// TwinCAT 3 PLC project PML_Base_Library
// Title: PML_Base_Library
// Company: SPT
// ProjectVersion: 0.1
// ProgramVersion: 3.1.4023.0
// libraries:
//   Tc2_Standard, * (Beckhoff Automation GmbH)
//   Tc2_System, * (Beckhoff Automation GmbH)
//   Tc3_EventLogger, * (Beckhoff Automation GmbH)
//   Tc3_PackML_V2, * (Beckhoff Automation GmbH)
// project tree:
//   Base/01_PML/01_Module/01_Base/01_GVL/ GVL_PML_Base.TcGVL
//   Base/01_PML/01_Module/01_Base/02_DUT/01_ENUM/ E_AlarmResponse.TcDUT, E_PMLUnitMode.TcDUT
//   Base/01_PML/01_Module/01_Base/02_DUT/02_STRUCT/ ST_PMLModuleBase_HMI.TcDUT, ST_PMLModuleBase_VISU.TcDUT, ST_PMLSubUnitInfoExt.TcDUT
//   Base/01_PML/01_Module/01_Base/03_ITFs/ ITF_PMLControl.TcIO, ITF_PMLModuleBase.TcIO
//   Base/01_PML/01_Module/01_Base/ FB_PMLModuleBase.TcPOU
//   Base/01_PML/01_Module/02_Events/ FB_PMLModeLogger.TcPOU, FB_PMLStateLogger.TcPOU
//   Base/01_PML/01_Module/03_PMLControl/03_ITFs/ ITF_PackML_ExternalControl.TcIO, ITF_PackML_ExternalControl_Simplified.TcIO
//   Base/01_PML/01_Module/03_PMLControl/ FB_ModuleExternalCommandControl.TcPOU, FB_PackML_ExternalControl.TcPOU, FB_PackML_PushButtonControl.TcPOU
//   Base/01_PML/01_Module/05_Visualizations/ V_MachineModule.TcVIS, V_Module.TcVIS
//   Base/01_PML/99_Templates/ FB_Module_TEMPLATE.TcPOU
//   Base/02_Component/ FB_ComponentBase.TcPOU, ITF_ComponentBase.TcIO, ST_ComponentBase_HMI.TcDUT
//   Base/03_Utilities/01_Events/ F_CreateAllEventsInClass.TcPOU, F_GetMaxSeverityRaised.TcPOU, F_RaiseAlarmAndSetFlags.TcPOU, F_RaiseAlarmWithStringParameters.TcPOU, F_RaiseAlarmWithStringsAndFlags.TcPOU
//   Base/03_Utilities/02_DataStructures/01_Tree/01_Tree_IndexBased/ FB_Tree_IndexBased.TcPOU, ITF_Tree_IndexBased.TcIO, ST_Tree_IndexBased_Node.TcDUT
//   Base/03_Utilities/02_DataStructures/02_FIFO/ FB_FIFO_ULINT_Array.TcPOU
//   Base/03_Utilities/03_Math/01_LREAL/ F_LREAL_RoundToPlace.TcPOU
//   / GlobalTextList.TcGTLO, Visualization Manager.TcVMO (not stored)

// ---- Base/01_PML/01_Module/01_Base/02_DUT/01_ENUM/E_AlarmResponse.TcDUT
{attribute 'qualified_only'}
{attribute 'strict'}
TYPE E_AlarmResponse :
(
	Abort_ImmediateError,
	Abort_Immediate,
	Stop_Immediate,
	Stop_Controlled,
	Hold_Immediate,
	Hold_Controlled,	
	Suspend_Immediate,
	Suspend_Controlled,
	NoResponse	
);
END_TYPE

// ---- Base/01_PML/01_Module/01_Base/02_DUT/01_ENUM/E_PMLUnitMode.TcDUT
{attribute 'qualified_only'}		//Note that this is not "Strict" since it needs to interact with the mode manager, which uses DINTs for mode
TYPE E_PMLUnitMode:
(
	ePMLUnitMode_Invalid 		:= 0,
	ePMLUnitMode_Production		:= 1,
	ePMLUnitMode_Maintenance	:= 2,
	ePMLUnitMode_Manual			:= 3
	// User defined modes
    (*ePMLUnitMode_SemiAutomatic  :=  4,
    ePMLUnitMode_DryRun         :=  5,
	ePMLUnitMode_Standalone		:=  6,
	ePMLUnitMode_Usermode4		:=  7,
	ePMLUnitMode_Usermode5 		:=  8,
	ePMLUnitMode_Usermode6 		:=  9,
	ePMLUnitMode_Usermode7 		:=  10 *)	
) DINT;
END_TYPE

// ---- Base/01_PML/01_Module/01_Base/02_DUT/02_STRUCT/ST_PMLModuleBase_HMI.TcDUT
TYPE ST_PMLModuleBase_HMI :
STRUCT
	bEnabled							: BOOL;					//Enables or disables the packml Machine of the module (prevents the module from going past idle)
	eMode								: E_PMLUnitMode;		//Current UnitMode of the module
	nModuleID							: UDINT;				//Unique identifying number for the module
	sModuleName							: STRING;				//Human-readable module name for user-side messaging
	eState								: Tc3_PackML_V2.E_PMLState;
	bLogStateChanges 					: BOOL := TRUE; 		//Toggle to permit or suppress state change logging (Should be tied to HMI setting to optionally reduce event logger clutter)
	bLogModeChanges 					: BOOL := TRUE; 		//Toggle to permit or suppress state change logging (Should be tied to HMI setting to optionally reduce event logger clutter)
	
	//Control information
	bHMIControlAvailable				: BOOL;		//Set TRUE *FROM PLC* when HMI requests can be processed
	bIncomingHMIRequest 				: BOOL;		//Pulses TRUE when an HMI request is issued
	bHMICommandConfirmation				: BOOL;		//Confirms receipt and subsequent processing of the command sent by the HMI
	
	bModeCommandHMIRequest				: BOOL;		//Pulses TRUE when an HMI mode change request is issued
	bStateCommandHMIRequest				: BOOL;		//Pulses TRUE when an HMI state change request is issued
	bEnableHMIRequest					: BOOL;		//HMI requests to enable the module
	bDisableHMIRequest 					: BOOL;		//HMI requests to disable the module
	bActivateStateLogHMIRequest			: BOOL;		//HMI requests to enable the module
	bDeactivateStateLogHMIRequest 		: BOOL;		//HMI requests to disable the module
	bActivateModeLogHMIRequest			: BOOL;		//HMI requests to enable the module
	bDeactivateModeLogHMIRequest 		: BOOL;		//HMI requests to disable the module
	eModeCommandHMIValue				: E_PMLUnitMode;
	eStateCommandHMIValue				: Tc3_PackML_V2.E_PMLCommand;
	a_sModeNames						: ARRAY[0..31] OF STRING;
	
END_STRUCT
END_TYPE

// ---- Base/01_PML/01_Module/01_Base/02_DUT/02_STRUCT/ST_PMLModuleBase_VISU.TcDUT
TYPE ST_PMLModuleBase_VISU :
STRUCT
	bEnabled			: BOOL;					//Enables or disables the packml Machine of the module (prevents the module from going past idle)
	eMode				: E_PMLUnitMode;		//Current UnitMode of the module
	nModuleID			: UDINT;					//Unique identifying number for the module
	sModuleName			: STRING;				//Human-readable module name for user-side messaging
	eState				: Tc3_PackML_V2.E_PMLState;
	
	//eModeCommandValue	: E_PMLUnitMode;
	///eStateCommandValue	: Tc3_PackML_V2.E_PMLCommand;
	bStartPressed		: BOOL;
	///bStartEnabled		: BOOL;
	bStopPressed		: BOOL;
	///bStopEnabled		: BOOL;
	bResetPressed		: BOOL;
	///bResetEnabled		: BOOL;
	bClearPressed		: BOOL;
	///bClearEnabled		: BOOL;	
	
	bAbortPressed		: BOOL;
	bHoldPressed		: BOOL;
	bUnholdPressed		: BOOL;
	bSuspendPressed		: BOOL;
	bUnsuspendPressed	: BOOL;
	
	// Mode things
	bProductionPressed	: BOOL;
	bMaintenancePressed	: BOOL;
	bManualPressed		: BOOL;
	
END_STRUCT
END_TYPE

// ---- Base/01_PML/01_Module/01_Base/02_DUT/02_STRUCT/ST_PMLSubUnitInfoExt.TcDUT
TYPE ST_PMLSubUnitInfoExt EXTENDS ST_PMLSubUnitInfo :	//Extended Struct of ST_PMLSubUnitInfo
STRUCT
	nModuleID 						: DINT; 				//Machine ID for messaging and Identification
	sModuleName						: STRING;				//Human readable machine name for messaging
	UnitModeCurrent					: E_PMLProtectedUnitMode;
	ActiveAlarm						: BOOL;
END_STRUCT
END_TYPE

// ---- Base/02_Component/ST_ComponentBase_HMI.TcDUT
TYPE ST_ComponentBase_HMI :
STRUCT
	//Status information
	bEnabled	: BOOL;
	bSimulate 	: BOOL;
	sName		: STRING;
	bActive		: BOOL;
	bError		: BOOL;
	nErrorID	: UDINT;
	
	//Control information
	bHMIControlAvailable	: BOOL;		//Set TRUE *FROM PLC* when HMI requests can be processed
	bIncomingHMIRequest 	: BOOL;		//Pulses TRUE when an HMI request is issued
	bHMICommandConfirmation	: BOOL;		//Confirms receipt and subsequent processing of the command sent by the HMI
	
	bEnableHMIRequest				: BOOL;		//HMI requests to enable the component
	bDisableHMIRequest 				: BOOL;		//HMI requests to disable the component
	bSimulateOperationHMIRequest 	: BOOL;		//HMI requests to change the component to simulation mode
	bStandardOperationHMIRequest	: BOOL;		//HMI requests to change the component to standard mode
	bResetHMIRequest				: BOOL;		//HMI requests to reset the component
	
END_STRUCT
END_TYPE

// ---- Base/03_Utilities/02_DataStructures/01_Tree/01_Tree_IndexBased/ST_Tree_IndexBased_Node.TcDUT
TYPE ST_Tree_IndexBased_Node :
STRUCT
	sName 		: STRING;
	nChildCount	: DINT;
	nParent		: DINT;
	a_nChildren	: ARRAY[0..15] OF DINT;
	nDepth		: DINT;
END_STRUCT
END_TYPE

// ---- Base/01_PML/01_Module/01_Base/01_GVL/GVL_PML_Base.TcGVL
///{attribute 'qualified_only'}
VAR_GLOBAL CONSTANT
	MAX_NO_OF_SUBMODULES			: UDINT := 20;
	MAX_NO_OF_COMPONENTS			: UDINT := 32;

	ePMLUNITMODEDEFAULT			: E_PMLUnitMode := E_PMLUnitMode.ePMLUnitMode_Production;
	ePMLSTATEDEFAULT			: E_PMLCommand := E_PMLCommand.ePMLCommand_Abort;

END_VAR

// ---- Base/01_PML/01_Module/01_Base/03_ITFs/ITF_PMLControl.TcIO
INTERFACE ITF_PMLControl

PROPERTY Mode : E_PMLUnitMode
GET
END_GET
END_PROPERTY

PROPERTY ModeCommand : DINT
SET
END_SET
END_PROPERTY

PROPERTY State : E_PMLState
GET
END_GET
END_PROPERTY

PROPERTY StateCommand : E_PMLCommand
SET
END_SET
END_PROPERTY

END_INTERFACE

// ---- Base/01_PML/01_Module/01_Base/03_ITFs/ITF_PMLModuleBase.TcIO
INTERFACE ITF_PMLModuleBase EXTENDS ITF_PMLControl

PROPERTY AncestorIDs : STRING
GET
END_GET
SET
END_SET
END_PROPERTY

PROPERTY CurrentAlarmSeverity :  TcEventSeverity
GET
END_GET
END_PROPERTY

METHOD CyclicLogic
END_METHOD

PROPERTY Enabled : BOOL
GET
END_GET
SET
END_SET
END_PROPERTY

PROPERTY LogModeChanges : BOOL
GET
END_GET
SET
END_SET
END_PROPERTY

PROPERTY LogStateChanges : BOOL
GET
END_GET
SET
END_SET
END_PROPERTY

PROPERTY MasterDataStructure_Adder :  ITF_Tree_IndexBased
GET
END_GET
SET
END_SET
END_PROPERTY

PROPERTY ModuleID : UDINT
GET
END_GET
SET
END_SET
END_PROPERTY

PROPERTY ModuleName : STRING
GET
END_GET
SET
END_SET
END_PROPERTY

PROPERTY ParentResponse_Critical : E_AlarmResponse
GET
END_GET
SET
END_SET
END_PROPERTY

PROPERTY ParentResponse_Error : E_AlarmResponse
GET
END_GET
SET
END_SET
END_PROPERTY

PROPERTY ParentResponse_Warning : E_AlarmResponse
GET
END_GET
SET
END_SET
END_PROPERTY

PROPERTY ParentResponseDef : ARRAY[0..4] OF E_AlarmResponse
GET
END_GET
SET
END_SET
END_PROPERTY

PROPERTY SimulateAllChildren : BOOL
GET
END_GET
SET
END_SET
END_PROPERTY

END_INTERFACE

// ---- Base/01_PML/01_Module/03_PMLControl/03_ITFs/ITF_PackML_ExternalControl.TcIO
INTERFACE ITF_PackML_ExternalControl EXTENDS ITF_PackML_ExternalControl_Simplified

PROPERTY Mode : DINT
GET
END_GET
SET
END_SET
END_PROPERTY

PROPERTY ModeCommand : DINT
GET
END_GET
SET
END_SET
END_PROPERTY

PROPERTY ModeCommandPulse : BOOL
GET
END_GET
SET
END_SET
END_PROPERTY

PROPERTY State : E_PMLState
GET
END_GET
SET
END_SET
END_PROPERTY

PROPERTY StateCommand : E_PMLCommand
GET
END_GET
SET
END_SET
END_PROPERTY

PROPERTY StateCommandPulse : BOOL
GET
END_GET
SET
END_SET
END_PROPERTY

END_INTERFACE

// ---- Base/01_PML/01_Module/03_PMLControl/03_ITFs/ITF_PackML_ExternalControl_Simplified.TcIO
INTERFACE ITF_PackML_ExternalControl_Simplified


PROPERTY ClearEnabled : BOOL
GET
END_GET
SET
END_SET
END_PROPERTY


PROPERTY ClearPressed : BOOL
GET
END_GET
SET
END_SET
END_PROPERTY

PROPERTY ResetEnabled : BOOL
GET
END_GET
SET
END_SET
END_PROPERTY

PROPERTY ResetPressed : BOOL
GET
END_GET
SET
END_SET
END_PROPERTY

PROPERTY StartEnabled : BOOL
GET
END_GET
SET
END_SET
END_PROPERTY

PROPERTY StartPressed : BOOL
GET
END_GET
SET
END_SET
END_PROPERTY

PROPERTY StopEnabled : BOOL
GET
END_GET
SET
END_SET
END_PROPERTY

PROPERTY StopPressed : BOOL
GET
END_GET
SET
END_SET
END_PROPERTY

END_INTERFACE

// ---- Base/02_Component/ITF_ComponentBase.TcIO
INTERFACE ITF_ComponentBase

PROPERTY Active : BOOL	//TRUE when the component is in motion or otherwise completing a commanded task
GET
END_GET
END_PROPERTY

METHOD AllowHMIControl : BOOL
VAR_INPUT
END_VAR
END_METHOD

METHOD BlockHMIControl : BOOL
VAR_INPUT
END_VAR
END_METHOD

PROPERTY CurrentAlarmSeverity : TcEventSeverity
GET
END_GET
END_PROPERTY

METHOD CyclicLogic : BOOL		//Should be called Externally akin to the PML Modules
END_METHOD

PROPERTY Enabled : BOOL	//Enables or disables the component
GET
END_GET
SET
END_SET
END_PROPERTY

PROPERTY Error : BOOL	//Boolean to signal that an error has ocurred
GET
END_GET
END_PROPERTY

PROPERTY ErrorID : UDINT	//Integer ID to identify the proper alarm to be posted from the parent module
GET
END_GET
SET
END_SET
END_PROPERTY

PROPERTY Name : STRING
GET
END_GET
SET
END_SET
END_PROPERTY

PROPERTY ParentResponseDefinitions : ARRAY[0..4] OF E_AlarmResponse
GET
END_GET
SET
END_SET
END_PROPERTY

PROPERTY Ready : BOOL
GET
END_GET
END_PROPERTY

METHOD Reset : BOOL
END_METHOD


PROPERTY Simulate : BOOL
GET
END_GET
SET
END_SET
END_PROPERTY

END_INTERFACE

// ---- Base/03_Utilities/02_DataStructures/01_Tree/01_Tree_IndexBased/ITF_Tree_IndexBased.TcIO
INTERFACE ITF_Tree_IndexBased

METHOD AddNodeAsChildByName : BOOL
VAR_INPUT
	sNewName 	: STRING;
	sParentName	: STRING;
END_VAR
END_METHOD

END_INTERFACE

// ---- Base/01_PML/01_Module/01_Base/FB_PMLModuleBase.TcPOU
FUNCTION_BLOCK ABSTRACT FB_PMLModuleBase IMPLEMENTS ITF_PMLModuleBase
VAR CONSTANT
	//Constant declarations
	PRODUCTION_DATA_ALARM_COUNT	: UDINT := 16;
END_VAR
VAR PERSISTENT
	//ITF_ProductionData internal variables
	tShiftLength: TIME := T#10M;
	nShiftProductionTarget	: DINT := 1000;
	fWarningMargin			: LREAL := 10;
	fProductionRate_Setpoint	: LREAL := 30;
	nRateAveragingCount		: DINT := 10;
END_VAR
VAR
	//ITF_PMLModuleBase internal property variables
	sAncestorIDs		: STRING;				//String concatenation of preceding parent IDs to prefix this module's ID
	bLogModeChanges 	: BOOL := TRUE; 		//Toggle to permit or suppress state change logging (Should be tied to HMI setting to optionally reduce event logger clutter)
	bLogStateChanges 	: BOOL := FALSE; 		//Toggle to permit or suppress state change logging (Should be tied to HMI setting to optionally reduce event logger clutter)
	nModuleID			: UDINT;					//Unique identifying number for the module
	sModuleName			: STRING;				//Human-readable module name for user-side messaging
	bEnabled			: BOOL := TRUE;			//Enables or disables the packml Machine of the module (prevents the module from going past idle)
	eModeCommand		: E_PMLUnitMode; 				//Current Commanded UnitMode of the module
	eStateCommand		: Tc3_PackML_V2.E_PMLCommand;
	eMode				: E_PMLUnitMode;		//Current UnitMode of the module
	eState				: Tc3_PackML_V2.E_PMLState;
	iMasterDataStructure_Adder : ITF_Tree_IndexBased;
	eCurrentAlarmSeverity		: TcEventSeverity;
	a_eParentFaultResponseDefinitions		: ARRAY[0..4] OF E_AlarmResponse := [	E_AlarmResponse.NoResponse,
																					E_AlarmResponse.NoResponse,
																					E_AlarmResponse.NoResponse,
																					E_AlarmResponse.Abort_ImmediateError,
																					E_AlarmResponse.Abort_ImmediateError];
	
	fbFIFO							: FB_FIFO_ULINT_Array;
	a_fbProductionDataAlarms		: ARRAY[1..PRODUCTION_DATA_ALARM_COUNT] OF FB_TcAlarm;
	fTemp : LREAL;



	//Communication Variables
	stPMLModuleBaseHMI	: ST_PMLModuleBase_HMI;		//Handles status and control communications with the HMI
	stPMLModuleBaseVISU	: ST_PMLModuleBase_VISU;	//Handles status and control communications with Visualizations
	fbExternalControl	: FB_ModuleExternalCommandControl;	//Handles commands from HMI/VISUS ^^ kind of overlaps with the structures above - TODO: Improve

	//Administration and Configuration Variables
	bInitialized 					: BOOL;					//TRUE when initialization code of the object is complete
	sID_Name						: STRING;				//"Module XX - 'Module Name' " Alarm and message utility phrase based off of nMachine ID and sMachineName
	
	//State and Mode control blocks
	fbModeManager 					: PML_UnitModeManager; 	//Manages operating mode transitions and rules
	fbStateMachine 					: PML_StateMachine; 	//Manages PackML state transitions
	fbCustomModes 					: PML_UnitModeConfig;	//Used to define custom machine modes if desired

	//State and Mode Status and Command variables
	sState							: STRING; 				//String representation of the current state
	eLastState						: E_PMLState;			//Last cycle PackML state
	eLastStateCommand				: E_PMLCommand;			//Previous received PackML state command
	eLastMode		 				: DINT;					//Last PackML mode 
	eLastModeCommand 				: E_PMLUnitMode;					//Previous received PackML mode command
	bStateTasksComplete				: BOOL := FALSE;					//All tasks to be performed at this program level are complete
	bNoStateTasksToComplete			: BOOL := TRUE;					//Indicates whether this stateneeds to perform tasks other than commanding its children
	bSubModulesReady				: BOOL;					//All submodules have reached the commanded state
	
	//Alarming and Logging variables - Some may or may not be necessary depending on final alarm system implementation ----------------------------------------------
	//These are for the newer TMC Excel import style alarm system
	a_fbPMLAlarms					: ARRAY[1..48] OF FB_TcAlarm;	//Array of alarms for PackML state and mode changes that exist in any PackML enabled module
	a_fbBaseAlarms					: ARRAY[1..32] OF FB_TcAlarm;		//Array of alarms for general module Alarms				
	fbPMLStateLogger				: FB_PMLStateLogger;				//Logs PackML state changes
	fbPMLModeLogger					: FB_PMLModeLogger;					//Logs PackML Mode changes

	// Alarm handling
	bActiveAlarm					: BOOL;					//module has an active alarm		TODO: Implement			
	bGlobalSafetyStatus				: BOOL;
	//********************************************************************************************************************
	// Sub Module variables
	// Used mostly for EMs and Machines, but ok for CM. They are just null	
	a_ITF_PackMLBase				: ARRAY[1..MAX_NO_OF_SUBMODULES] OF ITF_PMLModuleBase;	
	// Array of the PML sub unit info array used by the statemachine
	a_stPMLSubUnitInfo				: ARRAY[1..MAX_NO_OF_SUBMODULES] OF ST_PMLSubUnitInfo;
	nNumberOfSubModules				: UDINT := 0;	//calculated number of instantiated sub modules
	// This is the information for each module's submodules.
	PMLSubUnitInfoRef				: ST_PMLSubUnitInfoRef;				// Reference to the subunit information, used by the state machine
	//********************************************************************************************************************
	
	//Component variables - Allow iterative control of child components (Mostly used with Control Modules, but usable anywhere)
	a_ITF_Components				: ARRAY[1..MAX_NO_OF_COMPONENTS] OF ITF_ComponentBase;
	nNumberOfComponents				: UDINT := 0;	//calculated number of instantiated components
	
	//Miscellaneous Variables
	fLastProductionRate_Setpoint 	: LREAL;
	nIndex							: UDINT;		//Generic iteration value
	bSimulateAllChildren			: BOOL;
	a_sModeNames					: ARRAY[0..31] OF STRING;
	varInfo							: __SYSTEM.VAR_INFO;
	bReachedInitialDefaultStateAndMode	: BOOL;		//Toggles TRUE once a module has reached the default state and mode after startup, used to mute certain alarms during startup
	i: UDINT;
END_VAR

//*********************************************************
// !!!!! Code implementation only in CyclicLogic() method !!!!! 
//*********************************************************

METHOD Aborted
//*************************************************************************************************************************************************************************
//If you are about to write application specific code, note that any such code should exist within the "Application" directory using a Function Block that 'EXTENDS' this base Function Block!
//This particular method's functionality can be overriden in the extended block by creating a method of the same name, with desired functionality therein
//If the functionality of this base module is to be retained, but more functionality is desired, the extended method can contain a SUPER^.ThisMethodName(); call, which will call this code
//*************************************************************************************************************************************************************************

;
END_METHOD

METHOD AbortImmediate : BOOL
VAR_INPUT
END_VAR
eStateCommand := E_PMLCommand.ePMLCommand_Abort;
END_METHOD

METHOD AbortImmediateError : BOOL
VAR_INPUT
	sName		: STRING;
	bIsModule	: BOOL;
END_VAR
IF bIsModule THEN
	IF NOT a_fbBaseAlarms[E_BaseAlarms.SubModuleError].bRaised THEN
		F_RaiseAlarmWithStringParameters(a_fbBaseAlarms[E_BaseAlarms.SubModuleError],sModuleName,sName,'');
	END_IF
ELSE
	IF NOT a_fbBaseAlarms[E_BaseAlarms.ComponentError].bRaised THEN
		F_RaiseAlarmWithStringParameters(a_fbBaseAlarms[E_BaseAlarms.ComponentError],sModuleName,sName,'');
	END_IF
END_IF


eStateCommand := E_PMLCommand.ePMLCommand_Abort;
END_METHOD

METHOD Aborting
//*************************************************************************************************************************************************************************
//If you are about to write application specific code, note that any such code should exist within the "Application" directory using a Function Block that 'EXTENDS' this base Function Block!
//This particular method's functionality can be overriden in the extended block by creating a method of the same name, with desired functionality therein
//If the functionality of this base module is to be retained, but more functionality is desired, the extended method can contain a SUPER^.ThisMethodName(); call, which will call this code
//*************************************************************************************************************************************************************************

//Perform State tasks here
// Send abort command to all sub modules
FOR nIndex := 1 TO nNumberOfSubModules DO
	a_ITF_PackMLBase[nIndex].StateCommand:=ePMLCommand_Abort;
END_FOR

// All subunits in requested state?
bSubModulesReady := TRUE;

FOR nIndex := 1 TO nNumberOfSubModules DO
	bSubModulesReady := bSubModulesReady AND (a_ITF_PackMLBase[nIndex].State = ePMLState_Aborted);
END_FOR
IF bSubModulesReady AND (bStateTasksComplete OR bNoStateTasksToComplete) THEN
	bNoStateTasksToComplete := TRUE;
	bStateTasksComplete := FALSE;
	StateComplete();
END_IF
END_METHOD

METHOD AllowHMIControl : BOOL
VAR_INPUT
	bModuleOnly		: BOOL;	//If TRUE, only the PML module itself is controllable, If FALSE, all components become controllable as well
END_VAR
stPMLModuleBaseHMI.bHMIControlAvailable := TRUE;

IF bModuleOnly THEN
	FOR i := 1 TO nNumberOfComponents DO
		a_ITF_Components[i].BlockHMIControl();
	END_FOR
ELSE
	FOR i := 1 TO nNumberOfComponents DO
		a_ITF_Components[i].AllowHMIControl();
	END_FOR
END_IF
END_METHOD

PROPERTY AncestorIDs : STRING
GET
AncestorIDs := sAncestorIDs;
END_GET
SET
sAncestorIDs := AncestorIDs;
END_SET
END_PROPERTY

METHOD BlockHMIControl : BOOL
VAR_INPUT
END_VAR
stPMLModuleBaseHMI.bHMIControlAvailable := FALSE;

FOR i := 1 TO nNumberOfComponents DO
	a_ITF_Components[i].BlockHMIControl();
END_FOR
END_METHOD

METHOD Clearing
//*************************************************************************************************************************************************************************
//If you are about to write application specific code, note that any such code should exist within the "Application" directory using a Function Block that 'EXTENDS' this base Function Block!
//This particular method's functionality can be overriden in the extended block by creating a method of the same name, with desired functionality therein
//If the functionality of this base module is to be retained, but more functionality is desired, the extended method can contain a SUPER^.ThisMethodName(); call, which will call this code
//*************************************************************************************************************************************************************************

//Perform State tasks here
// Send clear command to all sub modules
FOR nIndex := 1 TO nNumberOfSubModules DO	
	a_ITF_PackMLBase[nIndex].StateCommand := ePMLCommand_Clear;
END_FOR

IF a_fbBaseAlarms[E_BaseAlarms.ComponentError].bRaised THEN
	a_fbBaseAlarms[E_BaseAlarms.ComponentError].Clear(0,0);
END_IF;

IF a_fbBaseAlarms[E_BaseAlarms.SubModuleError].bRaised THEN
	a_fbBaseAlarms[E_BaseAlarms.SubModuleError].Clear(0,0);
END_IF;


// All subunits in requested state?
bSubModulesReady	:= TRUE;
FOR nIndex:=1 TO nNumberOfComponents DO
	IF a_ITF_Components[nIndex].Error THEN
		a_ITF_Components[nIndex].Reset();
	END_IF
END_FOR

FOR nIndex:=1 TO nNumberOfComponents DO		
		bSubModulesReady := bSubModulesReady AND NOT a_ITF_Components[nIndex].Error;
END_FOR

FOR nIndex := 1 TO nNumberOfSubModules DO
	bSubModulesReady := bSubModulesReady AND (a_ITF_PackMLBase[nIndex].State = ePMLState_Stopped);
END_FOR
IF bSubModulesReady AND (bStateTasksComplete OR bNoStateTasksToComplete) THEN
	bNoStateTasksToComplete := TRUE;
	bStateTasksComplete := FALSE;
	StateComplete();
END_IF
END_METHOD

METHOD Complete
//*************************************************************************************************************************************************************************
//If you are about to write application specific code, note that any such code should exist within the "Application" directory using a Function Block that 'EXTENDS' this base Function Block!
//This particular method's functionality can be overriden in the extended block by creating a method of the same name, with desired functionality therein
//If the functionality of this base module is to be retained, but more functionality is desired, the extended method can contain a SUPER^.ThisMethodName(); call, which will call this code
//*************************************************************************************************************************************************************************

;
END_METHOD

METHOD Completing
//*************************************************************************************************************************************************************************
//If you are about to write application specific code, note that any such code should exist within the "Application" directory using a Function Block that 'EXTENDS' this base Function Block!
//This particular method's functionality can be overriden in the extended block by creating a method of the same name, with desired functionality therein
//If the functionality of this base module is to be retained, but more functionality is desired, the extended method can contain a SUPER^.ThisMethodName(); call, which will call this code
//*************************************************************************************************************************************************************************

//Perform State tasks here
// Send complete command to all sub modules
FOR nIndex := 1 TO nNumberOfSubModules DO
	a_ITF_PackMLBase[nIndex].StateCommand:=ePMLCommand_Complete;
END_FOR

// All subunits in requested state?
bSubModulesReady	:= TRUE;
FOR nIndex := 1 TO nNumberOfSubModules DO
	bSubModulesReady := bSubModulesReady AND (a_ITF_PackMLBase[nIndex].State = ePMLState_Complete);
END_FOR
IF bSubModulesReady AND (bStateTasksComplete OR bNoStateTasksToComplete) THEN
	bNoStateTasksToComplete := TRUE;
	bStateTasksComplete := FALSE;
	StateComplete();
END_IF
END_METHOD

METHOD ComponentMonitor : BOOL
VAR
	a_eAlarmResponses		: ARRAY[0..4] OF E_AlarmResponse;	//Temporary response array
END_VAR
FOR i:=1 TO nNumberOfComponents DO
	IF bSimulateAllChildren THEN
		a_ITF_Components[i].Simulate := TRUE;
	ELSE 
		a_ITF_Components[i].Simulate := FALSE;
	END_IF
	
	IF eMode = E_PMLUnitMode.ePMLUnitMode_Production THEN
		IF 		eState <> E_PMLState.ePMLState_Aborted
			AND eState <> E_PMLState.ePMLState_Aborting
			AND eState <> E_PMLState.ePMLState_Clearing
			AND eState <> E_PMLState.ePMLState_Stopped
			AND eState <> E_PMLState.ePMLState_Stopping
		THEN
			a_eAlarmResponses := a_ITF_Components[i].ParentResponseDefinitions;
			CASE a_eAlarmResponses[a_ITF_Components[i].CurrentAlarmSeverity] OF
				E_AlarmResponse.Abort_ImmediateError:
					AbortImmediateError(a_ITF_Components[i].Name, FALSE);
				E_AlarmResponse.Abort_Immediate:
					AbortImmediate();
				E_AlarmResponse.Stop_Immediate:
					StopImmediate();
				E_AlarmResponse.Stop_Controlled:
					StopControlled();
				E_AlarmResponse.Hold_Immediate:
					HoldImmediate();
				E_AlarmResponse.Suspend_Immediate:
					SuspendImmediate();
				E_AlarmResponse.Suspend_Controlled:
					SuspendControlled();
				E_AlarmResponse.NoResponse:
					;
			END_CASE
		ELSIF eState = E_PMLState.ePMLState_Stopped
			OR eState = E_PMLState.ePMLState_Stopping 
		THEN
			a_eAlarmResponses := a_ITF_Components[i].ParentResponseDefinitions;
			CASE a_eAlarmResponses[a_ITF_Components[i].CurrentAlarmSeverity] OF
				E_AlarmResponse.Abort_ImmediateError:
					AbortImmediateError(a_ITF_Components[i].Name, FALSE);
				E_AlarmResponse.Abort_Immediate:
					AbortImmediate();
				E_AlarmResponse.NoResponse:
					;
			END_CASE				
		END_IF
	END_IF		
END_FOR
END_METHOD

{attribute 'call_after_online_change_slot' := '<slot>'}
METHOD CreateEvents : BOOL
VAR_INPUT
END_VAR

VAR
END_VAR

F_CreateAllEventsInClass(	p_aAlarms := a_fbPMLAlarms,
							nClassSize := SIZEOF(TC_EVENTS.PMLAlarms),
							pInitEvent := ADR(TC_EVENTS.PMLAlarms.InitReferenceEvent),
							sPrefix := sID_Name);
							
F_CreateAllEventsInClass(	p_aAlarms := a_fbBaseAlarms,
							nClassSize := SIZEOF(TC_EVENTS.BaseAlarms),
							pInitEvent := ADR(TC_EVENTS.BaseAlarms.InitReferenceEvent),
							sPrefix := sID_Name);							
							
F_CreateAllEventsInClass(	p_aAlarms := a_fbProductionDataAlarms,
							nClassSize := SIZEOF(TC_EVENTS.ProductionData),
							pInitEvent := ADR(TC_EVENTS.ProductionData.InitReferenceEvent),
							sPrefix := sID_Name);
END_METHOD

PROPERTY CurrentAlarmSeverity : TcEventSeverity
GET
CurrentAlarmSeverity := eCurrentAlarmSeverity;
END_GET
END_PROPERTY

// 
// Cyclic Code
METHOD CyclicLogic
//*********************************************************
//If you are about to write actual machine implementation code, note that implementation code should exist within an implementation machine module block that extends this machine module base!
//*********************************************************

// First loop initialization code is triggered by highest level class
IF NOT bInitialized THEN			//Force initialization code of the object
	initialize();
	bInitialized := TRUE;
END_IF

//TODO: Condition state based on DEFAULT constant, right now it is a command, so a case statement translation to state would be necessary
IF NOT bReachedInitialDefaultStateAndMode AND eState = E_PMLState.ePMLState_Aborted AND eMode = ePMLUNITMODEDEFAULT THEN
	bReachedInitialDefaultStateAndMode := TRUE;
END_IF

//  call the subunits
FOR i := 1 TO nNumberOfSubModules DO	
	a_ITF_PackMLBase[i].CyclicLogic();								//Call the main cyclic loop of the subunits 
	a_stPMLSubUnitInfo[i].eState := a_ITF_PackMLBase[i].State;  	//Reflect the state of the subunits to the state machine of the module
END_FOR

FOR i:=1 TO nNumberOfComponents DO
	IF a_ITF_Components[i] <> 0 THEN
		a_ITF_Components[i].CyclicLogic();
	END_IF
END_FOR


// Mode control loop of the module
ModeControl();

// State control loop of the module
StateControl();

HMICommunication();
VISUCommunication();
fbExternalControl();
SubModuleMonitor();
ComponentMonitor();
HMIPermissions();

eCurrentAlarmSeverity := TcEventSeverity.Verbose;

eCurrentAlarmSeverity := F_GetMaxSeverityRaised(	a_fbAlarms := a_fbPMLAlarms,
													eCurrentSeverity := eCurrentAlarmSeverity);
eCurrentAlarmSeverity := F_GetMaxSeverityRaised(	a_fbAlarms := a_fbBaseAlarms,
													eCurrentSeverity := eCurrentAlarmSeverity);
END_METHOD

PROPERTY Enabled : BOOL
GET
Enabled := bEnabled;
END_GET
SET
bEnabled := Enabled;
END_SET
END_PROPERTY

METHOD Execute
//*************************************************************************************************************************************************************************
//If you are about to write application specific code, note that any such code should exist within the "Application" directory using a Function Block that 'EXTENDS' this base Function Block!
//This particular method's functionality can be overriden in the extended block by creating a method of the same name, with desired functionality therein
//If the functionality of this base module is to be retained, but more functionality is desired, the extended method can contain a SUPER^.ThisMethodName(); call, which will call this code
//*************************************************************************************************************************************************************************

;
END_METHOD

METHOD Held
//*************************************************************************************************************************************************************************
//If you are about to write application specific code, note that any such code should exist within the "Application" directory using a Function Block that 'EXTENDS' this base Function Block!
//This particular method's functionality can be overriden in the extended block by creating a method of the same name, with desired functionality therein
//If the functionality of this base module is to be retained, but more functionality is desired, the extended method can contain a SUPER^.ThisMethodName(); call, which will call this code
//*************************************************************************************************************************************************************************
END_METHOD

METHOD HMICommunication : BOOL
//Extend this method in extended FBs to communicate specific implementation data

//Process HMI requests
IF stPMLModuleBaseHMI.bIncomingHMIRequest AND NOT stPMLModuleBaseHMI.bHMICommandConfirmation THEN		//If a request has been issued by the HMI, and a previous request has not just E_SequenceState.Finished being processed
	
	IF stPMLModuleBaseHMI.bHMIControlAvailable THEN		//If the current conditions permit HMI control (Should be determined by the extended application components)
		IF stPMLModuleBaseHMI.bEnableHMIRequest THEN
			bEnabled := TRUE;
			stPMLModuleBaseHMI.bHMICommandConfirmation := TRUE;	//Confirm that the request has been processed
		END_IF
		IF stPMLModuleBaseHMI.bDisableHMIRequest THEN
			bEnabled := FALSE;
			stPMLModuleBaseHMI.bHMICommandConfirmation := TRUE;	//Confirm that the request has been processed
		END_IF
		IF stPMLModuleBaseHMI.bStateCommandHMIRequest THEN
			eStateCommand := stPMLModuleBaseHMI.eStateCommandHMIValue;
			//fbExternalControl.ExternalControlHMI.StateCommand := stPMLModuleBaseHMI.eStateCommandHMIValue;
			//fbExternalControl.ExternalControlHMI.StateCommandPulse := TRUE;
			stPMLModuleBaseHMI.bHMICommandConfirmation := TRUE;	//Confirm that the request has been processed
		END_IF
		IF stPMLModuleBaseHMI.bModeCommandHMIRequest THEN
			eModeCommand := stPMLModuleBaseHMI.eModeCommandHMIValue;
			//fbExternalControl.ExternalControlHMI.ModeCommand := stPMLModuleBaseHMI.eModeCommandHMIValue;
			//fbExternalControl.ExternalControlHMI.ModeCommandPulse := TRUE;
			stPMLModuleBaseHMI.bHMICommandConfirmation := TRUE;	//Confirm that the request has been processed
		END_IF
	END_IF
	
		//The following commands are always permissible, and are therefore not conditioned with bHMIControlAvailable
	IF stPMLModuleBaseHMI.bActivateStateLogHMIRequest THEN
		bLogStateChanges := TRUE;
		stPMLModuleBaseHMI.bHMICommandConfirmation := TRUE;	//Confirm that the request has been processed
	END_IF
	IF stPMLModuleBaseHMI.bDeactivateStateLogHMIRequest THEN
		bLogStateChanges := FALSE;
		stPMLModuleBaseHMI.bHMICommandConfirmation := TRUE;	//Confirm that the request has been processed
	END_IF
	IF stPMLModuleBaseHMI.bActivateModeLogHMIRequest THEN
		bLogModeChanges := TRUE;
		stPMLModuleBaseHMI.bHMICommandConfirmation := TRUE;	//Confirm that the request has been processed
	END_IF
	IF stPMLModuleBaseHMI.bDeactivateModeLogHMIRequest THEN
		bLogModeChanges := FALSE;
		stPMLModuleBaseHMI.bHMICommandConfirmation := TRUE;	//Confirm that the request has been processed
	END_IF		
END_IF


//Update HMI status info
stPMLModuleBaseHMI.bEnabled := bEnabled;
stPMLModuleBaseHMI.eMode := eMode;		//KAB eMode;
stPMLModuleBaseHMI.nModuleID := nModuleID;
stPMLModuleBaseHMI.sModuleName := sModuleName;
stPMLModuleBaseHMI.eState := eState;	//KAB eState;
stPMLModuleBaseHMI.bLogStateChanges := bLogStateChanges;
stPMLModuleBaseHMI.bLogModeChanges := bLogModeChanges;
stPMLModuleBaseHMI.a_sModeNames := a_sModeNames;
END_METHOD

PROPERTY HMIControlAvailable : BOOL
GET
HMIControlAvailable := stPMLModuleBaseHMI.bHMIControlAvailable;
END_GET
SET
stPMLModuleBaseHMI.bHMIControlAvailable := HMIControlAvailable;
END_SET
END_PROPERTY

METHOD HMIPermissions : BOOL
VAR_INPUT
END_VAR
//General Mode Based Monitoring and handling of HMI control
CASE eMode OF
//	====================================================================================================================================	
	E_PMLUnitMode.ePMLUnitMode_Production:			//=================================PRODUCTION MODE==================================
		CASE eState OF
			E_PMLState.ePMLState_Stopped:
				AllowHMIControl(bModuleOnly := TRUE);		//Allow control for recovery
			E_PMLState.ePMLState_Idle:
				BlockHMIControl();
			E_PMLState.ePMLState_Suspended:
				BlockHMIControl();
			E_PMLState.ePMLState_Execute:
				BlockHMIControl();
			E_PMLState.ePMLState_Aborted:
				AllowHMIControl(bModuleOnly := TRUE);		//Allow control for recovery
			E_PMLState.ePMLState_Held:
				AllowHMIControl(bModuleOnly := TRUE);		//Allow control for recovery
			E_PMLState.ePMLState_Complete:
				BlockHMIControl();
		END_CASE
		
//	====================================================================================================================================	
	E_PMLUnitMode.ePMLUnitMode_Manual:				//=================================MANUAL MODE======================================
		AllowHMIControl(bModuleOnly := FALSE);
//	====================================================================================================================================	
	E_PMLUnitMode.ePMLUnitMode_Maintenance:			//=================================MAINTENANCE MODE=================================
		AllowHMIControl(bModuleOnly := FALSE);	
END_CASE
END_METHOD

METHOD HoldControlled : BOOL
VAR_INPUT
END_VAR
END_METHOD

METHOD HoldImmediate : BOOL
VAR_INPUT
END_VAR
END_METHOD

METHOD Holding
//*************************************************************************************************************************************************************************
//If you are about to write application specific code, note that any such code should exist within the "Application" directory using a Function Block that 'EXTENDS' this base Function Block!
//This particular method's functionality can be overriden in the extended block by creating a method of the same name, with desired functionality therein
//If the functionality of this base module is to be retained, but more functionality is desired, the extended method can contain a SUPER^.ThisMethodName(); call, which will call this code
//*************************************************************************************************************************************************************************

//Perform State tasks here
// Send hold command to all sub modules
FOR nIndex := 1 TO nNumberOfSubModules DO
	a_ITF_PackMLBase[nIndex].StateCommand:=ePMLCommand_Hold;
END_FOR

// All subunits in requested state?
bSubModulesReady	:= TRUE;
FOR nIndex := 1 TO nNumberOfSubModules DO
	bSubModulesReady := bSubModulesReady AND (a_ITF_PackMLBase[nIndex].State = ePMLState_Held);
END_FOR
IF bSubModulesReady AND (bStateTasksComplete OR bNoStateTasksToComplete) THEN
	bNoStateTasksToComplete := TRUE;
	bStateTasksComplete := FALSE;
	StateComplete();
END_IF
END_METHOD

METHOD Idle
//*************************************************************************************************************************************************************************
//If you are about to write application specific code, note that any such code should exist within the "Application" directory using a Function Block that 'EXTENDS' this base Function Block!
//This particular method's functionality can be overriden in the extended block by creating a method of the same name, with desired functionality therein
//If the functionality of this base module is to be retained, but more functionality is desired, the extended method can contain a SUPER^.ThisMethodName(); call, which will call this code
//*************************************************************************************************************************************************************************
END_METHOD

METHOD initialize
VAR
	i : UDINT;
END_VAR
sID_Name := CONCAT(CONCAT(CONCAT(CONCAT(CONCAT('Module ', sAncestorIDs), UDINT_TO_STRING(nModuleID)), ' - '), sModuleName), ' '); 	//Creates a utility string for alarms and other messaging that reads (example text) - "Module 10 - Main Casepacker" to be followed by the alarm or message info
CreateEvents();

// Figure out how many Submodules were instantiated - they should be from 1 to X and not skip any indices.
nNumberOfSubModules := 0;
FOR i:=1 TO MAX_NO_OF_SUBMODULES DO
	IF a_ITF_PackMLBase[i] <> 0 THEN
		IF iMasterDataStructure_Adder <> 0 THEN
			iMasterDataStructure_Adder.AddNodeAsChildByName(sNewName := a_ITF_PackMLBase[i].ModuleName, sParentName := ModuleName);
		ELSIF NOT a_fbBaseAlarms[E_BaseAlarms.InvalidInterface].bRaised THEN
			varInfo :=  __VARINFO(iMasterDataStructure_Adder);
			F_RaiseAlarmWithStringParameters(a_fbBaseAlarms[E_BaseAlarms.InvalidInterface], sModuleName, varInfo.Symbol, '');	
		END_IF
		nNumberOfSubModules:=nNumberOfSubModules+1;
		
		a_ITF_PackMLBase[i].AncestorIDs := CONCAT(CONCAT(AncestorIDs, DINT_TO_STRING(ModuleID)), '_');
		a_ITF_PackMLBase[i].MasterDataStructure_Adder 	:= iMasterDataStructure_Adder;
		IF a_ITF_PackMLBase[i].ModuleID = 0 THEN	//If the ID was not manually initialized to anything at declaration, automatically assign it an ID
			a_ITF_PackMLBase[i].ModuleID := i;
		END_IF
	END_IF
END_FOR

nNumberOfComponents := 0;
FOR i:=1 TO MAX_NO_OF_COMPONENTS DO
	IF a_ITF_Components[i] <> 0 THEN

		a_ITF_Components[i].Name := CONCAT(CONCAT(sModuleName,' '),a_ITF_Components[i].Name);	//Add the name of the module as a prefix to the name given in the declaration initialization
		
		IF iMasterDataStructure_Adder <> 0 THEN
			iMasterDataStructure_Adder.AddNodeAsChildByName(sNewName := a_ITF_Components[i].Name, sParentName := ModuleName);
		ELSIF NOT a_fbBaseAlarms[E_BaseAlarms.InvalidInterface].bRaised THEN
			varInfo :=  __VARINFO(iMasterDataStructure_Adder);
			F_RaiseAlarmWithStringParameters(a_fbBaseAlarms[E_BaseAlarms.InvalidInterface], sModuleName, varInfo.Symbol, '');	
		END_IF
		nNumberOfComponents:=nNumberOfComponents+1;
	END_IF
END_FOR

fbExternalControl.Module := THIS^;

// <BASIC INITIALIZATION CODE, DO NOT CHANGE>
// Initialize subunit overview used by state machine
PMLSubUnitInfoRef.ArraySize := SIZEOF(a_stPMLSubUnitInfo);
PMLSubUnitInfoRef.NoOfSubUnits := nNumberOfSubModules;
PMLSubUnitInfoRef.pArray := ADR(a_stPMLSubUnitInfo);
// Point the state machine to the locally defined subunit info 
//fbStateMachine.stSubUnitInfoRef := PMLSubUnitInfoRef;
// <\BASIC INITIALIZATION CODE, DO NOT CHANGE>

// Activate all subunits by default, or change accordingly
FOR i:=1 TO nNumberOfSubModules DO
	a_stPMLSubUnitInfo[i].Active	:= TRUE;					// Follows Main State Machine
END_FOR

FOR i:=1 TO nNumberOfComponents DO
	IF a_ITF_Components[i] <> 0 THEN
		a_ITF_Components[i].Enabled := TRUE;
	END_IF
END_FOR
END_METHOD

PROPERTY LogModeChanges : BOOL
GET
LogModeChanges:= bLogModeChanges;
END_GET
SET
bLogModeChanges := LogModeChanges;
END_SET
END_PROPERTY

PROPERTY LogStateChanges : BOOL
GET
LogStateChanges:= bLogStateChanges;
END_GET
SET
bLogStateChanges := LogStateChanges;
END_SET
END_PROPERTY

PROPERTY MasterDataStructure_Adder :  ITF_Tree_IndexBased
GET
MasterDataStructure_Adder := iMasterDataStructure_Adder;
END_GET
SET
iMasterDataStructure_Adder := MasterDataStructure_Adder;
END_SET
END_PROPERTY

PROPERTY Mode : E_PMLUnitMode
GET
Mode := eMode;
END_GET
END_PROPERTY

PROPERTY ModeCommand : DINT
SET
eModeCommand := ModeCommand;
END_SET
END_PROPERTY

METHOD PRIVATE ModeControl
VAR
	i					: UDINT;
END_VAR
//On startup, Mode is invalid, set it to production
IF eMode = E_PMLUnitMode.ePMLUnitMode_Invalid 		THEN 
	fbModeManager.bExecute 		:= TRUE; 
	eModeCommand			 	:= ePMLUNITMODEDEFAULT; 
	eLastModeCommand 			:= eModeCommand;
//If mode is valid and the command has changed, attempt to change modes
ELSIF eModeCommand <> eLastModeCommand 					THEN
	//DONKEY : logging to be implemented
	fbModeManager.bExecute 		:= TRUE;
	eLastModeCommand 			:= eModeCommand;
END_IF

//Handles mode changes based on eModeCommand and the state transition rules defined in the pre-defined protected modes or custom modes
fbModeManager(
	eModeCommand			:= eModeCommand, 
	eState					:= eState, 			
	eModeStatus				=> eMode, 
	bDone					=> , 
	bError					=> , 
	nErrorId				=> 
	);
	
IF fbModeManager.bError AND bReachedInitialDefaultStateAndMode THEN
	IF NOT a_fbPMLAlarms[E_PMLAlarms.ModeCommandInvalid].bRaised THEN
		a_fbPMLAlarms[E_PMLAlarms.ModeCommandInvalid].Raise(0);
	END_IF
ELSIF a_fbPMLAlarms[E_PMLAlarms.ModeCommandInvalid].bRaised THEN
	a_fbPMLAlarms[E_PMLAlarms.ModeCommandInvalid].Clear(0,0);
END_IF

// Reset mode control command
fbModeManager.bExecute 		:= FALSE;

//If PackML mode has changed
IF fbModeManager.eModeStatus <> eLastMode  THEN 
	eLastMode := fbModeManager.eModeStatus; 
	//If state change logging is not suppressed
 	IF bLogModeChanges THEN 
		fbPMLModeLogger(
			a_fbPMLAlarms := a_fbPMLAlarms,
			sModulePrefix := sID_Name,
			Mode := fbModeManager.eModeStatus);	
	END_IF	
	// Change SubModules
	FOR i := 1 TO nNumberOfSubModules DO
		a_ITF_PackMLBase[i].ModeCommand := fbModeManager.eModeStatus;		//Call the SetMode loop of the subunits 
	END_FOR

END_IF
END_METHOD

PROPERTY ModuleID : UDINT
GET
ModuleID := nModuleID;
END_GET
SET
nModuleID := ModuleID;
END_SET
END_PROPERTY

PROPERTY ModuleName : STRING
GET
ModuleName := sModuleName;
END_GET
SET
sModuleName := ModuleName;
END_SET
END_PROPERTY

PROPERTY ParentResponse_Critical : E_AlarmResponse
GET
ParentResponse_Critical := a_eParentFaultResponseDefinitions[TcEventSeverity.Critical];
END_GET
SET
a_eParentFaultResponseDefinitions[TcEventSeverity.Critical] := ParentResponse_Critical;
END_SET
END_PROPERTY

PROPERTY ParentResponse_Error : E_AlarmResponse
GET
ParentResponse_Error := a_eParentFaultResponseDefinitions[TcEventSeverity.Error];
END_GET
SET
a_eParentFaultResponseDefinitions[TcEventSeverity.Error] := ParentResponse_Error;
END_SET
END_PROPERTY

PROPERTY ParentResponse_Warning : E_AlarmResponse
GET
ParentResponse_Warning := a_eParentFaultResponseDefinitions[TcEventSeverity.Warning];
END_GET
SET
a_eParentFaultResponseDefinitions[TcEventSeverity.Warning] := ParentResponse_Warning;
END_SET
END_PROPERTY

PROPERTY ParentResponseDef : ARRAY[0..4] OF E_AlarmResponse
GET
ParentResponseDef[TcEventSeverity.Verbose] := a_eParentFaultResponseDefinitions[TcEventSeverity.Verbose];
ParentResponseDef[TcEventSeverity.Info] := a_eParentFaultResponseDefinitions[TcEventSeverity.Info];
ParentResponseDef[TcEventSeverity.Warning] := a_eParentFaultResponseDefinitions[TcEventSeverity.Warning];
ParentResponseDef[TcEventSeverity.Error] := a_eParentFaultResponseDefinitions[TcEventSeverity.Error];
ParentResponseDef[TcEventSeverity.Critical] := a_eParentFaultResponseDefinitions[TcEventSeverity.Critical];
END_GET
SET
a_eParentFaultResponseDefinitions[TcEventSeverity.Verbose] := ParentResponseDef[TcEventSeverity.Verbose];
a_eParentFaultResponseDefinitions[TcEventSeverity.Info] := ParentResponseDef[TcEventSeverity.Info];
a_eParentFaultResponseDefinitions[TcEventSeverity.Warning] := ParentResponseDef[TcEventSeverity.Warning];
a_eParentFaultResponseDefinitions[TcEventSeverity.Error] := ParentResponseDef[TcEventSeverity.Error];
a_eParentFaultResponseDefinitions[TcEventSeverity.Critical] := ParentResponseDef[TcEventSeverity.Critical];
END_SET
END_PROPERTY

METHOD Resetting
//*************************************************************************************************************************************************************************
//If you are about to write application specific code, note that any such code should exist within the "Application" directory using a Function Block that 'EXTENDS' this base Function Block!
//This particular method's functionality can be overriden in the extended block by creating a method of the same name, with desired functionality therein
//If the functionality of this base module is to be retained, but more functionality is desired, the extended method can contain a SUPER^.ThisMethodName(); call, which will call this code
//*************************************************************************************************************************************************************************

//Perform State tasks here
// Send clear/reset command to all sub modules
//As long as this module is in the "Resetting" state, it will attempt to get all modules to Idle by sending abort, clear, and reset commands as appropriate to its children until they do
FOR nIndex := 1 TO nNumberOfSubModules DO
	IF a_ITF_PackMLBase[nIndex].State=ePMLState_Stopped OR a_ITF_PackMLBase[nIndex].State=ePMLState_Complete THEN
		a_ITF_PackMLBase[nIndex].StateCommand:=ePMLCommand_Reset;
	ELSIF a_ITF_PackMLBase[nIndex].State=ePMLState_Aborted THEN
		a_ITF_PackMLBase[nIndex].StateCommand:=ePMLCommand_Clear;
	ELSIF a_ITF_PackMLBase[nIndex].State=ePMLState_Clearing OR a_ITF_PackMLBase[nIndex].State=ePMLState_Stopping 
		OR a_ITF_PackMLBase[nIndex].State=ePMLState_Resetting OR a_ITF_PackMLBase[nIndex].State=ePMLState_Idle THEN
		;
	ELSE
		a_ITF_PackMLBase[nIndex].StateCommand:=ePMLCommand_Abort;
	END_IF
END_FOR

FOR nIndex:=1 TO nNumberOfComponents DO
	IF NOT a_ITF_Components[nIndex].Enabled THEN
		a_ITF_Components[nIndex].Enabled := TRUE;
	END_IF
END_FOR


// All subunits in requested state?
bSubModulesReady	:= TRUE;

FOR nIndex:=1 TO nNumberOfComponents DO		
	bSubModulesReady := bSubModulesReady AND a_ITF_Components[nIndex].Ready;
END_FOR

FOR nIndex := 1 TO nNumberOfSubModules DO
	bSubModulesReady := bSubModulesReady AND (a_ITF_PackMLBase[nIndex].State = ePMLState_Idle);
END_FOR
IF bSubModulesReady AND (bStateTasksComplete OR bNoStateTasksToComplete) THEN
	bNoStateTasksToComplete := TRUE;
	bStateTasksComplete := FALSE;
	StateComplete();
END_IF
END_METHOD

PROPERTY SimulateAllChildren : BOOL
GET
SimulateAllChildren := bSimulateAllChildren;
END_GET
SET
bSimulateAllChildren := SimulateAllChildren;
END_SET
END_PROPERTY

METHOD Starting
//*************************************************************************************************************************************************************************
//If you are about to write application specific code, note that any such code should exist within the "Application" directory using a Function Block that 'EXTENDS' this base Function Block!
//This particular method's functionality can be overriden in the extended block by creating a method of the same name, with desired functionality therein
//If the functionality of this base module is to be retained, but more functionality is desired, the extended method can contain a SUPER^.ThisMethodName(); call, which will call this code
//*************************************************************************************************************************************************************************

//Perform State tasks here
// Send start command to all sub modules
FOR nIndex := 1 TO nNumberOfSubModules DO
	a_ITF_PackMLBase[nIndex].StateCommand:=ePMLCommand_Start;
END_FOR

// All subunits in requested state?
bSubModulesReady	:= TRUE; 
FOR nIndex := 1 TO nNumberOfSubModules DO
	bSubModulesReady := bSubModulesReady AND (a_ITF_PackMLBase[nIndex].State = ePMLState_Execute);
END_FOR 
IF bSubModulesReady AND (bStateTasksComplete OR bNoStateTasksToComplete) THEN
	bNoStateTasksToComplete := TRUE;
	bStateTasksComplete := FALSE;
	StateComplete();
END_IF
END_METHOD

PROPERTY State : Tc3_PackML_V2.E_PMLState
GET
State := eState;
END_GET
END_PROPERTY

PROPERTY StateCommand : Tc3_PackML_V2.E_PMLCommand
SET
IF 	eMode <> E_PMLUnitMode.ePMLUnitMode_Invalid 	AND
 	eState <> E_PMLState.ePMLState_Undefined 			THEN 
	eStateCommand := StateCommand;
END_IF
END_SET
END_PROPERTY

METHOD StateComplete
//*************************************************************************************************************************************************************************
//If you are about to write application specific code, note that any such code should exist within the "Application" directory using a Function Block that 'EXTENDS' this base Function Block!
//This particular method's functionality can be overriden in the extended block by creating a method of the same name, with desired functionality therein
//If the functionality of this base module is to be retained, but more functionality is desired, the extended method can contain a SUPER^.ThisMethodName(); call, which will call this code
//*************************************************************************************************************************************************************************

fbStateMachine.M_StateComplete();
END_METHOD

METHOD PRIVATE StateControl
//On startup, state is invalid, set it to default
IF eState = E_PMLState.ePMLState_Undefined 				AND 
	eMode <> E_PMLUnitMode.ePMLUnitMode_Invalid 	THEN 
	eStateCommand 	:= ePMLSTATEDEFAULT; 
END_IF

//Call PackML state machine	
fbStateMachine(
	eMode				:= eMode, 
	eCommand			:= eStateCommand, 
	stSubUnitInfoRef	:= ,
	stOptions			:= , 
	eState				=> eState, 
	sState 				=> sState, 
	bError				=> , 
	nErrorID			=> );

//If PackML state has changed
IF eState <> eLastState  THEN 
	eLastState := eState; 
	bNoStateTasksToComplete := TRUE;
END_IF 
	
IF bReachedInitialDefaultStateAndMode THEN
	//Log appropriate state changes
	fbPMLStateLogger(
		a_fbPMLAlarms := a_fbPMLAlarms, 
		sModulePrefix := SID_Name, 
		eState := eState,
		bLogAllChanges := bLogStateChanges);	
END_IF

// Call appropriate method depending on current PackML state
CASE eState OF
	E_PMLState.ePMLState_Undefined:
		Undefined();
	E_PMLState.ePMLState_Clearing:
		Clearing();
	E_PMLState.ePMLState_Stopped:
		Stopped();
	E_PMLState.ePMLState_Starting:
		Starting();
	E_PMLState.ePMLState_Idle:
		Idle();
	E_PMLState.ePMLState_Suspended:
		Suspended();
	E_PMLState.ePMLState_Execute:
		Execute();
	E_PMLState.ePMLState_Stopping:
		Stopping();
	E_PMLState.ePMLState_Aborting:
		Aborting();
	E_PMLState.ePMLState_Aborted:
		Aborted();
	E_PMLState.ePMLState_Holding:
		Holding();
	E_PMLState.ePMLState_Held:
		Held();
	E_PMLState.ePMLState_Unholding:
		Unholding();
	E_PMLState.ePMLState_Suspending:
		Suspending();
	E_PMLState.ePMLState_Unsuspending:
		Unsuspending();
	E_PMLState.ePMLState_Resetting:   	
		Resetting();
	E_PMLState.ePMLState_Completing:
		Completing();
	E_PMLState.ePMLState_Complete:
		Complete();
END_CASE
END_METHOD

METHOD StopControlled : BOOL
VAR_INPUT
END_VAR
END_METHOD

METHOD StopImmediate : BOOL
VAR_INPUT
END_VAR
eStateCommand := E_PMLCommand.ePMLCommand_Stop;
END_METHOD

METHOD Stopped
//*************************************************************************************************************************************************************************
//If you are about to write application specific code, note that any such code should exist within the "Application" directory using a Function Block that 'EXTENDS' this base Function Block!
//This particular method's functionality can be overriden in the extended block by creating a method of the same name, with desired functionality therein
//If the functionality of this base module is to be retained, but more functionality is desired, the extended method can contain a SUPER^.ThisMethodName(); call, which will call this code
//*************************************************************************************************************************************************************************
END_METHOD

METHOD Stopping
//*************************************************************************************************************************************************************************
//If you are about to write application specific code, note that any such code should exist within the "Application" directory using a Function Block that 'EXTENDS' this base Function Block!
//This particular method's functionality can be overriden in the extended block by creating a method of the same name, with desired functionality therein
//If the functionality of this base module is to be retained, but more functionality is desired, the extended method can contain a SUPER^.ThisMethodName(); call, which will call this code
//*************************************************************************************************************************************************************************

//Perform State tasks here
// Send stop command to all sub modules
FOR nIndex := 1 TO nNumberOfSubModules DO
	a_ITF_PackMLBase[nIndex].StateCommand:=ePMLCommand_Stop;
END_FOR

// All subunits in requested state?
bSubModulesReady	:= TRUE;
FOR nIndex := 1 TO nNumberOfSubModules DO
	bSubModulesReady := bSubModulesReady AND (a_ITF_PackMLBase[nIndex].State = ePMLState_Stopped OR a_ITF_PackMLBase[nIndex].State = ePMLState_Aborted);
END_FOR
IF bSubModulesReady AND (bStateTasksComplete OR bNoStateTasksToComplete) THEN
	bNoStateTasksToComplete := TRUE;
	bStateTasksComplete := FALSE;
	StateComplete();
END_IF
END_METHOD

METHOD SubModuleMonitor : BOOL
VAR
	a_eAlarmResponses		: ARRAY[0..4] OF E_AlarmResponse;	//Temporary response array	
END_VAR

FOR i := 1 TO nNumberOfSubModules DO
	
	IF bSimulateAllChildren THEN
		a_ITF_PackMLBase[i].SimulateAllChildren := TRUE;
	ELSE
		a_ITF_PackMLBase[i].SimulateAllChildren := FALSE;
	END_IF

	
	IF eMode = E_PMLUnitMode.ePMLUnitMode_Production THEN		
		IF 		eState <> E_PMLState.ePMLState_Aborted
			AND eState <> E_PMLState.ePMLState_Aborting
			AND eState <> E_PMLState.ePMLState_Clearing
			AND eState <> E_PMLState.ePMLState_Stopped
			AND eState <> E_PMLState.ePMLState_Stopping
		THEN
			a_eAlarmResponses := a_ITF_PackMLBase[i].ParentResponseDef;
			CASE a_eAlarmResponses[a_ITF_PackMLBase[i].CurrentAlarmSeverity] OF
				E_AlarmResponse.Abort_ImmediateError:
					AbortImmediateError(a_ITF_PackMLBase[i].ModuleName, TRUE);
				E_AlarmResponse.Abort_Immediate:
					AbortImmediate();
				E_AlarmResponse.Stop_Immediate:
					StopImmediate();
				E_AlarmResponse.Stop_Controlled:
					StopControlled();
				E_AlarmResponse.Hold_Immediate:
					HoldImmediate();
				E_AlarmResponse.Suspend_Immediate:
					SuspendImmediate();
				E_AlarmResponse.Suspend_Controlled:
					SuspendControlled();
				E_AlarmResponse.NoResponse:
					;
			END_CASE
		ELSIF eState = E_PMLState.ePMLState_Stopped
			OR eState = E_PMLState.ePMLState_Stopping 
		THEN
			a_eAlarmResponses := a_ITF_PackMLBase[i].ParentResponseDef;
			CASE a_eAlarmResponses[a_ITF_PackMLBase[i].CurrentAlarmSeverity] OF
				E_AlarmResponse.Abort_ImmediateError:
					AbortImmediateError(a_ITF_PackMLBase[i].ModuleName, TRUE);
				E_AlarmResponse.Abort_Immediate:
					AbortImmediate();
				E_AlarmResponse.NoResponse:
					;
			END_CASE				
		END_IF
	END_IF
END_FOR
END_METHOD

METHOD SuspendControlled : BOOL
VAR_INPUT
END_VAR
END_METHOD

METHOD Suspended
//*************************************************************************************************************************************************************************
//If you are about to write application specific code, note that any such code should exist within the "Application" directory using a Function Block that 'EXTENDS' this base Function Block!
//This particular method's functionality can be overriden in the extended block by creating a method of the same name, with desired functionality therein
//If the functionality of this base module is to be retained, but more functionality is desired, the extended method can contain a SUPER^.ThisMethodName(); call, which will call this code
//*************************************************************************************************************************************************************************
END_METHOD

METHOD SuspendImmediate : BOOL
VAR_INPUT
END_VAR
END_METHOD

METHOD Suspending
//*************************************************************************************************************************************************************************
//If you are about to write application specific code, note that any such code should exist within the "Application" directory using a Function Block that 'EXTENDS' this base Function Block!
//This particular method's functionality can be overriden in the extended block by creating a method of the same name, with desired functionality therein
//If the functionality of this base module is to be retained, but more functionality is desired, the extended method can contain a SUPER^.ThisMethodName(); call, which will call this code
//*************************************************************************************************************************************************************************

//Perform State tasks here
// Send suspend command to all sub modules
FOR nIndex := 1 TO nNumberOfSubModules DO
	a_ITF_PackMLBase[nIndex].StateCommand:=ePMLCommand_Suspend;
END_FOR

// All subunits in requested state?
bSubModulesReady	:= TRUE;
FOR nIndex := 1 TO nNumberOfSubModules DO
	bSubModulesReady := bSubModulesReady AND (a_ITF_PackMLBase[nIndex].State = ePMLState_Suspended);
END_FOR
IF bSubModulesReady AND (bStateTasksComplete OR bNoStateTasksToComplete) THEN
	bNoStateTasksToComplete := TRUE;
	bStateTasksComplete := FALSE;
	StateComplete();
END_IF
END_METHOD

PROPERTY TargetProductionRate : LREAL
GET
TargetProductionRate := fProductionRate_Setpoint;
END_GET
SET
fProductionRate_Setpoint := TargetProductionRate;
END_SET
END_PROPERTY

METHOD Undefined
//*************************************************************************************************************************************************************************
//If you are about to write application specific code, note that any such code should exist within the "Application" directory using a Function Block that 'EXTENDS' this base Function Block!
//This particular method's functionality can be overriden in the extended block by creating a method of the same name, with desired functionality therein
//If the functionality of this base module is to be retained, but more functionality is desired, the extended method can contain a SUPER^.ThisMethodName(); call, which will call this code
//*************************************************************************************************************************************************************************
END_METHOD

METHOD Unholding
//*************************************************************************************************************************************************************************
//If you are about to write application specific code, note that any such code should exist within the "Application" directory using a Function Block that 'EXTENDS' this base Function Block!
//This particular method's functionality can be overriden in the extended block by creating a method of the same name, with desired functionality therein
//If the functionality of this base module is to be retained, but more functionality is desired, the extended method can contain a SUPER^.ThisMethodName(); call, which will call this code
//*************************************************************************************************************************************************************************

//Perform State tasks here
// Send unhold command to all sub modules
FOR nIndex := 1 TO nNumberOfSubModules DO
	a_ITF_PackMLBase[nIndex].StateCommand:=ePMLCommand_Unhold;
END_FOR

// All subunits in requested state?
bSubModulesReady	:= TRUE;
FOR nIndex := 1 TO nNumberOfSubModules DO
	bSubModulesReady := bSubModulesReady AND (a_ITF_PackMLBase[nIndex].State = ePMLState_Execute);
END_FOR
IF bSubModulesReady AND (bStateTasksComplete OR bNoStateTasksToComplete) THEN
	bNoStateTasksToComplete := TRUE;
	bStateTasksComplete := FALSE;
	StateComplete();
END_IF
END_METHOD

METHOD Unsuspending
//*************************************************************************************************************************************************************************
//If you are about to write application specific code, note that any such code should exist within the "Application" directory using a Function Block that 'EXTENDS' this base Function Block!
//This particular method's functionality can be overriden in the extended block by creating a method of the same name, with desired functionality therein
//If the functionality of this base module is to be retained, but more functionality is desired, the extended method can contain a SUPER^.ThisMethodName(); call, which will call this code
//*************************************************************************************************************************************************************************

//Perform State tasks here
// Send unsuspend command to all sub modules
FOR nIndex := 1 TO nNumberOfSubModules DO
	a_ITF_PackMLBase[nIndex].StateCommand:=ePMLCommand_Unsuspend;
END_FOR

// All subunits in requested state?
bSubModulesReady	:= TRUE;
FOR nIndex := 1 TO nNumberOfSubModules DO
	bSubModulesReady := bSubModulesReady AND (a_ITF_PackMLBase[nIndex].State = ePMLState_Execute);
END_FOR
IF bSubModulesReady AND (bStateTasksComplete OR bNoStateTasksToComplete) THEN
	bNoStateTasksToComplete := TRUE;
	bStateTasksComplete := FALSE;
	StateComplete();
END_IF
END_METHOD

METHOD VISUCommunication : BOOL
VAR_INPUT
END_VAR

fbExternalControl.ExternalControlVISU.ClearPressed := stPMLModuleBaseVISU.bClearPressed;
fbExternalControl.ExternalControlVISU.ResetPressed := stPMLModuleBaseVISU.bResetPressed;
fbExternalControl.ExternalControlVISU.StartPressed := stPMLModuleBaseVISU.bStartPressed;
fbExternalControl.ExternalControlVISU.StopPressed := stPMLModuleBaseVISU.bStopPressed;


//Update VISU status info
stPMLModuleBaseVISU.bEnabled := bEnabled;
stPMLModuleBaseVISU.eMode := eMode;		
stPMLModuleBaseVISU.nModuleID := nModuleID;
stPMLModuleBaseVISU.sModuleName := sModuleName;
stPMLModuleBaseVISU.eState := eState;	

// Mode logic here.  Only taking the button from the visualizations
IF stPMLModuleBaseVISU.bProductionPressed AND eMode <> E_PMLUnitMode.ePMLUnitMode_Production THEN
	fbExternalControl.ExternalControlVISU.ModeCommand := E_PMLUnitMode.ePMLUnitMode_Production;
	fbExternalControl.ExternalControlVISU.ModeCommandPulse := TRUE;
END_IF
IF stPMLModuleBaseVISU.bMaintenancePressed AND eMode <> E_PMLUnitMode.ePMLUnitMode_Maintenance THEN
	fbExternalControl.ExternalControlVISU.ModeCommand := E_PMLUnitMode.ePMLUnitMode_Maintenance;
	fbExternalControl.ExternalControlVISU.ModeCommandPulse := TRUE;
END_IF
IF stPMLModuleBaseVISU.bManualPressed AND eMode <> E_PMLUnitMode.ePMLUnitMode_Manual THEN
	fbExternalControl.ExternalControlVISU.ModeCommand := E_PMLUnitMode.ePMLUnitMode_Manual;
	fbExternalControl.ExternalControlVISU.ModeCommandPulse := TRUE;
END_IF

// Extra buttons from Visu here for state changes than the standard 4
// Abort
IF stPMLModuleBaseVISU.bAbortPressed THEN
	CASE eState OF
		ePMLState_Aborted,
		ePMLState_Aborting:
			// DO Nothing
	ELSE
		fbExternalControl.ExternalControlVISU.StateCommand := E_PMLCommand.ePMLCommand_Abort;
		fbExternalControl.ExternalControlVISU.StateCommandPulse := TRUE;	
	END_CASE
END_IF

// Hold
IF stPMLModuleBaseVISU.bHoldPressed THEN
	IF eState = ePMLState_Execute THEN
		fbExternalControl.ExternalControlVISU.StateCommand := E_PMLCommand.ePMLCommand_Hold;
		fbExternalControl.ExternalControlVISU.StateCommandPulse := TRUE;	
	END_IF
END_IF

// unHold
IF stPMLModuleBaseVISU.bUnholdPressed THEN
	IF eState = ePMLState_Held THEN
		fbExternalControl.ExternalControlVISU.StateCommand := E_PMLCommand.ePMLCommand_Unhold;
		fbExternalControl.ExternalControlVISU.StateCommandPulse := TRUE;	
	END_IF
END_IF

// Suspend
IF stPMLModuleBaseVISU.bSuspendPressed THEN
	IF eState = ePMLState_Execute THEN
		fbExternalControl.ExternalControlVISU.StateCommand := E_PMLCommand.ePMLCommand_Suspend;
		fbExternalControl.ExternalControlVISU.StateCommandPulse := TRUE;	
	END_IF
END_IF

// unSuspend
IF stPMLModuleBaseVISU.bUnsuspendPressed THEN
	IF eState = ePMLState_Suspended THEN
		fbExternalControl.ExternalControlVISU.StateCommand := E_PMLCommand.ePMLCommand_Unsuspend;
		fbExternalControl.ExternalControlVISU.StateCommandPulse := TRUE;	
	END_IF
END_IF
END_METHOD

END_FUNCTION_BLOCK

// ---- Base/03_Utilities/02_DataStructures/02_FIFO/FB_FIFO_ULINT_Array.TcPOU
FUNCTION_BLOCK FB_FIFO_ULINT_Array
VAR_IN_OUT
	a_FIFO		: ARRAY [*] OF ULINT;
END_VAR
VAR_OUTPUT
END_VAR
VAR
	nEntryCount		: DINT;
END_VAR

METHOD AddEntry : BOOL
VAR_INPUT
	nEntry		: ULINT;
END_VAR
VAR
	i : DINT;
END_VAR
IF (LOWER_BOUND(a_FIFO, 1) + nEntryCount - 1) > UPPER_BOUND(a_FIFO, 1) THEN
	AddEntry := FALSE;		//FIFO is full
ELSE
	FOR i := UPPER_BOUND(a_FIFO,1) - 1 TO LOWER_BOUND(a_FIFO,1) BY -1 DO
		a_FIFO[i+1] := a_FIFO[i];
	END_FOR
	
	a_FIFO[LOWER_BOUND(a_FIFO,1)] := nEntry;
	
	nEntryCount := nEntryCount + 1;
	AddEntry := TRUE;
END_IF
END_METHOD

PROPERTY EntryCount : DINT
GET
EntryCount := nEntryCount;
END_GET
END_PROPERTY

PROPERTY LastInValue : ULINT
GET
IF nEntryCount = 0 THEN
	LastInValue := 0;
ELSE
	LastInValue := a_FIFO[LOWER_BOUND(a_FIFO,1)];
END_IF
END_GET
END_PROPERTY

PROPERTY NextOutValue : ULINT
GET
IF nEntryCount = 0 THEN
	NextOutValue := 0;
ELSE
	NextOutValue := a_FIFO[LOWER_BOUND(a_FIFO,1) + nEntryCount - 1];
END_IF
END_GET
END_PROPERTY

METHOD RemoveEntry : BOOL
VAR_INPUT
END_VAR
IF nEntryCount = 0 THEN
	RemoveEntry := FALSE;
ELSE
	IF (LOWER_BOUND(a_FIFO,1) + nEntryCount - 1) <= UPPER_BOUND(a_FIFO,1) THEN
		a_FIFO[LOWER_BOUND(a_FIFO,1) + nEntryCount - 1] := 0;
		nEntryCount := nEntryCount - 1; 
		RemoveEntry := TRUE;
	END_IF
END_IF
END_METHOD

END_FUNCTION_BLOCK

// ---- Base/01_PML/01_Module/03_PMLControl/FB_ModuleExternalCommandControl.TcPOU
FUNCTION_BLOCK FB_ModuleExternalCommandControl
VAR_INPUT
END_VAR
VAR_OUTPUT
END_VAR
VAR
	ipModulePackMLBase			: ITF_PMLModuleBase;
	
	fbHMIControl				: FB_PackML_ExternalControl;
	fbVISUControl				: FB_PackML_ExternalControl;
	fbPushButtonControl			: FB_PackML_PushButtonControl;
			
	a_iExternalControlSources	: ARRAY[1..3] OF ITF_PackML_ExternalControl := [fbHMIControl,fbVISUControl,fbPushButtonControl];	//Add more control sources as desired
	
	i : DINT;
END_VAR

FOR i := 1 TO 3 DO		//TODO: Make Dynamic through constant declaration or otherwise
	
	IF a_iExternalControlSources[i].ModeCommandPulse THEN
		ipModulePackMLBase.ModeCommand := a_iExternalControlSources[i].ModeCommand;
		a_iExternalControlSources[i].ModeCommandPulse := FALSE;
	END_IF
	
	IF a_iExternalControlSources[i].StateCommandPulse THEN
		ipModulePackMLBase.StateCommand := a_iExternalControlSources[i].StateCommand;
		a_iExternalControlSources[i].StateCommandPulse := FALSE;
	END_IF
	
	a_iExternalControlSources[i].Mode := ipModulePackMLBase.Mode;
	a_iExternalControlSources[i].State := ipModulePackMLBase.State;
END_FOR

fbHMIControl();
fbVISUControl();
///fbPushButtonControl();

PROPERTY ExternalControlHMI : ITF_PackML_ExternalControl
GET
ExternalControlHMI := a_iExternalControlSources[1];
END_GET
END_PROPERTY

PROPERTY ExternalControlVISU : ITF_PackML_ExternalControl
GET
ExternalControlVISU := a_iExternalControlSources[2];
END_GET
END_PROPERTY

PROPERTY Module : ITF_PMLModuleBase
GET
Module := ipModulePackMLBase;
END_GET
SET
ipModulePackMLBase := Module;
END_SET
END_PROPERTY

END_FUNCTION_BLOCK

// ---- Base/01_PML/01_Module/03_PMLControl/FB_PackML_ExternalControl.TcPOU
FUNCTION_BLOCK FB_PackML_ExternalControl IMPLEMENTS ITF_PackML_ExternalControl
VAR_INPUT
END_VAR
VAR_OUTPUT
END_VAR
VAR
	nMode				: DINT;
	nModeCommand		: DINT;
	bModeCommandPulse	: BOOL;
	eState				: Tc3_PackML_V2.E_PMLState;
	eStateCommand		: Tc3_PackML_V2.E_PMLCommand;
	bStateCommandPulse	: BOOL;
	
	bStartPressed		: BOOL;
	bStartEnabled		: BOOL;
	bStopPressed		: BOOL;
	bStopEnabled		: BOOL;
	bResetPressed		: BOOL;
	bResetEnabled		: BOOL;
	bClearPressed		: BOOL;
	bClearEnabled		: BOOL;	
	
END_VAR

//Handle button presses
IF bStartPressed THEN
	IF eState = Tc3_PackML_V2.E_PMLState.ePMLState_Idle THEN
		eStateCommand := Tc3_PackML_V2.E_PMLCommand.ePMLCommand_Start;
		bStateCommandPulse := TRUE;
	ELSIF eState = Tc3_PackML_V2.E_PMLState.ePMLState_Held THEN
		eStateCommand := Tc3_PackML_V2.E_PMLCommand.ePMLCommand_Unhold;
		bStateCommandPulse := TRUE;
	END_IF
	bStartPressed := FALSE;
END_IF

IF bStopPressed THEN
	eStateCommand := Tc3_PackML_V2.E_PMLCommand.ePMLCommand_Stop;
	bStateCommandPulse := TRUE;
	bStopPressed := FALSE;
END_IF

IF bResetPressed THEN
	eStateCommand := Tc3_PackML_V2.E_PMLCommand.ePMLCommand_Reset;
	bStateCommandPulse := TRUE;
	bResetPressed := FALSE;
END_IF

IF bClearPressed THEN
	eStateCommand := Tc3_PackML_V2.E_PMLCommand.ePMLCommand_Clear;
	bStateCommandPulse := TRUE;
	bClearPressed := FALSE;
END_IF

//Handle enabling of the Start button
IF 		eState = Tc3_PackML_V2.E_PMLState.ePMLState_Idle
	OR	eState = Tc3_PackML_V2.E_PMLState.ePMLState_Held 	THEN
	bStartEnabled := TRUE;
ELSE
	bStartEnabled := FALSE;
END_IF

//Handle enabling of the Stop button
IF 		eState <> Tc3_PackML_V2.E_PMLState.ePMLState_Stopped
	AND	eState <> Tc3_PackML_V2.E_PMLState.ePMLState_Clearing
	AND	eState <> Tc3_PackML_V2.E_PMLState.ePMLState_Aborted
	AND	eState <> Tc3_PackML_V2.E_PMLState.ePMLState_Aborting
	AND	eState <> Tc3_PackML_V2.E_PMLState.ePMLState_Undefined 	THEN
	bStopEnabled := TRUE;
ELSE
	bStopEnabled := FALSE;
END_IF

//Handle enabling of the Reset button
IF 		eState = Tc3_PackML_V2.E_PMLState.ePMLState_Complete
	OR	eState = Tc3_PackML_V2.E_PMLState.ePMLState_Stopped 	THEN
	bResetEnabled := TRUE;
ELSE
	bResetEnabled := FALSE;
END_IF

//Handle enabling of the Clear button
IF 		eState = Tc3_PackML_V2.E_PMLState.ePMLState_Aborted	THEN
	bClearEnabled := TRUE;
ELSE
	bClearEnabled := FALSE;
END_IF


// Handle mode changes


PROPERTY ClearEnabled : BOOL
GET
ClearEnabled := bClearEnabled;
END_GET
SET
bClearEnabled := ClearEnabled;
END_SET
END_PROPERTY


PROPERTY ClearPressed : BOOL
GET
ClearPressed := bClearPressed;
END_GET
SET
bClearPressed := ClearPressed;
END_SET
END_PROPERTY

PROPERTY Mode : DINT
GET
Mode := nMode;
END_GET
SET
nMode := Mode;
END_SET
END_PROPERTY


PROPERTY ModeCommand : DINT
GET
ModeCommand := nModeCommand;
END_GET
SET
nModeCommand := ModeCommand;
END_SET
END_PROPERTY


PROPERTY ModeCommandPulse : BOOL
GET
ModeCommandPulse := bModeCommandPulse;
END_GET
SET
bModeCommandPulse := ModeCommandPulse;
END_SET
END_PROPERTY


PROPERTY ResetEnabled : BOOL
GET
ResetEnabled := bResetEnabled;
END_GET
SET
bResetEnabled := ResetEnabled;
END_SET
END_PROPERTY


PROPERTY ResetPressed : BOOL
GET
bResetPressed := ResetPressed;
END_GET
SET
bResetPressed := ResetPressed;
END_SET
END_PROPERTY


PROPERTY StartEnabled : BOOL
GET
StartEnabled := bStartEnabled;
END_GET
SET
bStartEnabled := StartEnabled;
END_SET
END_PROPERTY


PROPERTY StartPressed : BOOL
GET
StartPressed := bStartPressed;
END_GET
SET
bStartPressed := StartPressed;
END_SET
END_PROPERTY


PROPERTY State : Tc3_PackML_V2.E_PMLState
GET
State := eState;
END_GET
SET
eState := State;
END_SET
END_PROPERTY


PROPERTY StateCommand : Tc3_PackML_V2.E_PMLCommand
GET
StateCommand := eStateCommand;
END_GET
SET
eStateCommand := StateCommand;
END_SET
END_PROPERTY


PROPERTY StateCommandPulse : BOOL
GET
StateCommandPulse := bStateCommandPulse;
END_GET
SET
bStateCommandPulse := StateCommandPulse;
END_SET
END_PROPERTY


PROPERTY StopEnabled : BOOL
GET
StopEnabled := bStopEnabled;
END_GET
SET
bStopEnabled := StopEnabled;
END_SET
END_PROPERTY


PROPERTY StopPressed : BOOL
GET
StopPressed := bStopPressed;
END_GET
SET
bStopPressed := StopPressed;
END_SET
END_PROPERTY

END_FUNCTION_BLOCK

// ---- Base/01_PML/01_Module/03_PMLControl/FB_PackML_PushButtonControl.TcPOU
FUNCTION_BLOCK FB_PackML_PushButtonControl EXTENDS FB_PackML_ExternalControl
VAR_INPUT
END_VAR
VAR_OUTPUT
END_VAR
VAR
	bStartButton	AT %I* : BOOL;	//Tie to hardware start pushbutton
	//TODO: add other buttons
END_VAR

//TODO: implement button control

END_FUNCTION_BLOCK

// ---- Base/01_PML/01_Module/02_Events/FB_PMLStateLogger.TcPOU
FUNCTION_BLOCK FB_PMLStateLogger
VAR_IN_OUT
	a_fbPMLAlarms			: ARRAY[1..48] OF FB_TcAlarm;		//Array of alarms for Core PackML events that exist in any PackML enabled module
END_VAR
VAR_INPUT
	sModulePrefix : STRING;	//Prefix String for all state change events (Typically the ID and Name of the module in some concatenated form)
	eState	: E_PMLState;	//Current PML state of the module
	bLogAllChanges	: BOOL := TRUE; //If TRUE, all state change events will be logged, regardless of severity, otherwise info alarms are ignored
END_VAR
VAR_OUTPUT
END_VAR
VAR
	eLastState : E_PMLState := E_PMLState.ePMLState_Aborted;		//Saves the previous state each time the block is run
	refTempAlarm : REFERENCE TO FB_TcAlarm;		//Temporary reference that makes severity checking simpler vs individually checking each change alarm within the case statement
END_VAR

IF eState <> eLastState THEN		//If state has changed
	CASE eState OF		//Get the stored alarm that corresponds to the newly entered state and save its reference temporarily
		E_PMLState.ePMLState_Starting:
			refTempAlarm REF= a_fbPMLAlarms[E_PMLAlarms.StateStartingEnter];
		E_PMLState.ePMLState_Execute:
			refTempAlarm REF= a_fbPMLAlarms[E_PMLAlarms.StateExecuteEnter];
		E_PMLState.ePMLState_Completing:
			refTempAlarm REF= a_fbPMLAlarms[E_PMLAlarms.StateCompletingEnter];
		E_PMLState.ePMLState_Complete:
			refTempAlarm REF= a_fbPMLAlarms[E_PMLAlarms.StateCompleteEnter];
		E_PMLState.ePMLState_Resetting:
			refTempAlarm REF= a_fbPMLAlarms[E_PMLAlarms.StateResettingEnter];
		E_PMLState.ePMLState_Idle:
			refTempAlarm REF= a_fbPMLAlarms[E_PMLAlarms.StateIdleEnter];
		E_PMLState.ePMLState_Holding:
			refTempAlarm REF= a_fbPMLAlarms[E_PMLAlarms.StateHoldingEnter];
		E_PMLState.ePMLState_Held:
			refTempAlarm REF= a_fbPMLAlarms[E_PMLAlarms.StateHeldEnter];
		E_PMLState.ePMLState_Unholding:
			refTempAlarm REF= a_fbPMLAlarms[E_PMLAlarms.StateUnholdingEnter];
		E_PMLState.ePMLState_Suspending:
			refTempAlarm REF= a_fbPMLAlarms[E_PMLAlarms.StateSuspendingEnter];
		E_PMLState.ePMLState_Suspended:
			refTempAlarm REF= a_fbPMLAlarms[E_PMLAlarms.StateSuspendedEnter];
		E_PMLState.ePMLState_Unsuspending:
			refTempAlarm REF= a_fbPMLAlarms[E_PMLAlarms.StateUnsuspendingEnter];
		E_PMLState.ePMLState_Stopping:
			refTempAlarm REF= a_fbPMLAlarms[E_PMLAlarms.StateStoppingEnter];
		E_PMLState.ePMLState_Stopped:
			refTempAlarm REF= a_fbPMLAlarms[E_PMLAlarms.StateStoppedEnter];
		E_PMLState.ePMLState_Aborting:
			refTempAlarm REF= a_fbPMLAlarms[E_PMLAlarms.StateAbortingEnter];
		E_PMLState.ePMLState_Aborted:
			refTempAlarm REF= a_fbPMLAlarms[E_PMLAlarms.StateAbortedEnter];
		E_PMLState.ePMLState_Clearing:
			refTempAlarm REF= a_fbPMLAlarms[E_PMLAlarms.StateClearingEnter];
		E_PMLState.ePMLState_Undefined:
			refTempAlarm REF= a_fbPMLAlarms[E_PMLAlarms.StateUndefinedEnter];
	END_CASE
	
	//If the FB is set to log all changes, log the change, otherwise check the severity of the alarm and log it if it exceeds 'info' severity
	IF bLogAllChanges OR (refTempAlarm.eSeverity <> TcEventSeverity.Info AND refTempAlarm.eSeverity <> TcEventSeverity.Verbose) THEN
		refTempAlarm.Raise(0);
	END_IF
	
	CASE eLastState OF	//Clear the previous state's event (Events will remain 'Raised' as long as the module remains in that state)
		E_PMLState.ePMLState_Starting:
			a_fbPMLAlarms[E_PMLAlarms.StateStartingEnter].Clear(0,0);
		E_PMLState.ePMLState_Execute:
			a_fbPMLAlarms[E_PMLAlarms.StateExecuteEnter].Clear(0,0);
		E_PMLState.ePMLState_Completing:
			a_fbPMLAlarms[E_PMLAlarms.StateCompletingEnter].Clear(0,0);
		E_PMLState.ePMLState_Complete:
			a_fbPMLAlarms[E_PMLAlarms.StateCompleteEnter].Clear(0,0);
		E_PMLState.ePMLState_Resetting:
			a_fbPMLAlarms[E_PMLAlarms.StateResettingEnter].Clear(0,0);
		E_PMLState.ePMLState_Idle:
			a_fbPMLAlarms[E_PMLAlarms.StateIdleEnter].Clear(0,0);
		E_PMLState.ePMLState_Holding:
			a_fbPMLAlarms[E_PMLAlarms.StateHoldingEnter].Clear(0,0);
		E_PMLState.ePMLState_Held:
			a_fbPMLAlarms[E_PMLAlarms.StateHeldEnter].Clear(0,0);
		E_PMLState.ePMLState_Unholding:
			a_fbPMLAlarms[E_PMLAlarms.StateUnholdingEnter].Clear(0,0);
		E_PMLState.ePMLState_Suspending:
			a_fbPMLAlarms[E_PMLAlarms.StateSuspendingEnter].Clear(0,0);
		E_PMLState.ePMLState_Suspended:
			a_fbPMLAlarms[E_PMLAlarms.StateSuspendedEnter].Clear(0,0);
		E_PMLState.ePMLState_Unsuspending:
			a_fbPMLAlarms[E_PMLAlarms.StateUnsuspendingEnter].Clear(0,0);
		E_PMLState.ePMLState_Stopping:
			a_fbPMLAlarms[E_PMLAlarms.StateStoppingEnter].Clear(0,0);
		E_PMLState.ePMLState_Stopped:
			a_fbPMLAlarms[E_PMLAlarms.StateStoppedEnter].Clear(0,0);
		E_PMLState.ePMLState_Aborting:
			a_fbPMLAlarms[E_PMLAlarms.StateAbortingEnter].Clear(0,0);
		E_PMLState.ePMLState_Aborted:
			a_fbPMLAlarms[E_PMLAlarms.StateAbortedEnter].Clear(0,0);
		E_PMLState.ePMLState_Clearing:
			a_fbPMLAlarms[E_PMLAlarms.StateClearingEnter].Clear(0,0);
		E_PMLState.ePMLState_Undefined:
			a_fbPMLAlarms[E_PMLAlarms.StateUndefinedEnter].Clear(0,0);

	END_CASE
	eLastState := eState;	//Store previous state
END_IF

END_FUNCTION_BLOCK

// ---- Base/01_PML/01_Module/02_Events/FB_PMLModeLogger.TcPOU
FUNCTION_BLOCK FB_PMLModeLogger
VAR_IN_OUT
	a_fbPMLAlarms			: ARRAY[1..48] OF FB_TcAlarm;		//Array of alarms for Core PackML events that exist in any PackML enabled module
END_VAR
VAR_INPUT
	sModulePrefix : STRING;	//Prefix String for any
	///State	: E_PMLState;
	Mode : DINT;
END_VAR
VAR_OUTPUT
END_VAR
VAR
	lastMode : DINT;
END_VAR

IF Mode <> lastMode THEN
	CASE Mode OF
		E_PMLUnitMode.ePMLUnitMode_Invalid:
			a_fbPMLAlarms[E_PMLAlarms.ModeInvalidEnter].Raise(0);
		E_PMLUnitMode.ePMLUnitMode_Production:	
			a_fbPMLAlarms[E_PMLAlarms.ModeProductionEnter].Raise(0);
		E_PMLUnitMode.ePMLUnitMode_Maintenance:
			a_fbPMLAlarms[E_PMLAlarms.ModeMaintenanceEnter].Raise(0);
		E_PMLUnitMode.ePMLUnitMode_Manual:
			a_fbPMLAlarms[E_PMLAlarms.ModeManualEnter].Raise(0);
	END_CASE
	
	CASE lastMode OF
		E_PMLUnitMode.ePMLUnitMode_Invalid:
			a_fbPMLAlarms[E_PMLAlarms.ModeInvalidEnter].Clear(0,0);
		E_PMLUnitMode.ePMLUnitMode_Production:	
			a_fbPMLAlarms[E_PMLAlarms.ModeProductionEnter].Clear(0,0);
		E_PMLUnitMode.ePMLUnitMode_Maintenance:
			a_fbPMLAlarms[E_PMLAlarms.ModeMaintenanceEnter].Clear(0,0);
		E_PMLUnitMode.ePMLUnitMode_Manual:
			a_fbPMLAlarms[E_PMLAlarms.ModeManualEnter].Clear(0,0);
	END_CASE
	lastMode := Mode;
END_IF

END_FUNCTION_BLOCK

// ---- Base/03_Utilities/01_Events/F_RaiseAlarmWithStringParameters.TcPOU
FUNCTION F_RaiseAlarmWithStringParameters : BOOL
VAR_IN_OUT
	fbAlarm			: FB_TcAlarm;	//Alarm to be raised
END_VAR
VAR_INPUT
	sString_1	: STRING;
	sString_2	: STRING;
	sString_3	: STRING;
END_VAR

fbAlarm.ipArguments.Clear();

IF sString_1 <> '' THEN
	fbAlarm.ipArguments.AddString(sString_1);
END_IF
IF sString_2 <> '' THEN
	fbAlarm.ipArguments.AddString(sString_2);
END_IF
IF sString_3 <> '' THEN
	fbAlarm.ipArguments.AddString(sString_3);
END_IF

fbAlarm.Raise(0);

END_FUNCTION

// ---- Base/03_Utilities/01_Events/F_CreateAllEventsInClass.TcPOU
FUNCTION F_CreateAllEventsInClass : BOOL
VAR_IN_OUT
	p_aAlarms : ARRAY[*] OF FB_TcAlarm;		//Array of Alarms to be defined
END_VAR
VAR_INPUT
	nClassSize : DINT;
	pInitEvent : POINTER TO TcEventEntry;	//Address of first event in Event Class (Should be the InitReferenceEvent)
	sPrefix	: STRING;	//String Prefix for the Event Message -- Usually the Module ID and Name
END_VAR
VAR
	i : DINT;
	nEventSize : DINT;
	numberOfEvents : DINT;
	pEvent	: POINTER TO TcEventEntry;
END_VAR

nEventSize := SIZEOF(pInitEvent^);
numberOfEvents := nClassSize/nEventSize;

FOR i := LOWER_BOUND(p_aAlarms,1) TO UPPER_BOUND(p_aAlarms,1) DO
	IF i > numberOfEvents THEN
		EXIT;
	ELSE
		pEvent := pInitEvent + ((i - 1) * nEventSize);
		p_aAlarms[i].CreateEx(stEventEntry := pEvent^, 0,0);
		p_aAlarms[i].ipArguments.AddString(sPrefix);
	END_IF
END_FOR

END_FUNCTION

// ---- Base/03_Utilities/01_Events/F_GetMaxSeverityRaised.TcPOU
FUNCTION F_GetMaxSeverityRaised : TcEventSeverity
VAR_IN_OUT
	a_fbAlarms			: ARRAY[*] OF FB_TcAlarm;
END_VAR
VAR_INPUT
	eCurrentSeverity	: TcEventSeverity;
END_VAR
VAR
	i					: DINT;
END_VAR


FOR i := LOWER_BOUND(a_fbAlarms, 1) TO UPPER_BOUND(a_fbAlarms, 1) DO
	IF a_fbAlarms[i].bRaised AND (a_fbAlarms[i].eSeverity > eCurrentSeverity) THEN
		eCurrentSeverity := a_fbAlarms[i].eSeverity;
	END_IF
END_FOR

F_GetMaxSeverityRaised := eCurrentSeverity;

END_FUNCTION

// ---- Base/01_PML/99_Templates/FB_Module_TEMPLATE.TcPOU
FUNCTION_BLOCK FB_Module_TEMPLATE EXTENDS FB_PMLModuleBase
VAR
	//Define the Sub modules here for this module. (If any)  Also set the Interfaces in the initialize method.
	(*fbSubModule1				: FB_ApplicationModule_TEMPLATE := (ModuleName :=  'Test Module 1');
	*)
	(*fbSubModule2				: FB_ApplicationModule_TEMPLATE := (ModuleName :=  'Test Module 2');
	*)
	//temporary array of module base interfaces to be copied over to the base class a_itfPackMLBase variable
	a_ITF_PackMLBase_init		: ARRAY[1..MAX_NO_OF_SUBMODULES] OF ITF_PMLModuleBase := [(*	fbSubModule1,
																							 	fbSubModule2*)];

	//Define the components here for this module. (If any) Also set the Interfaces in the initialize method.
	(*fbComponent1				: FB_ComponentBase (Extension):= (Name := 'Test Component 1');
	*)
	(*fbComponent2				: FB_ComponentBase (Extension):= (Name := 'Test Component 2');
	*)	
	//temporary array of module base interfaces to be copied over to the base class a_itfPackMLBase variable
	a_ITF_Components_init		: ARRAY[1..GVL_PML_Base.MAX_NO_OF_COMPONENTS ] OF ITF_ComponentBase := [(*	fbComponent1,
																											fbComponent2*)];
	
END_VAR

//*********************************************************
//Body of block is not called by base code, only implement application
//code in CyclicUpdate or in methods called by it or its subcalls
//*********************************************************

METHOD Aborted
CASE eMode OF
//	====================================================================PRODUCTION MODE=========================================================	
	E_PMLUnitMode.ePMLUnitMode_Production:			
		;
//	====================================================================MANUAL MODE=============================================================	
	E_PMLUnitMode.ePMLUnitMode_Manual:				
		;
//	=====================================================================MAINTENANCE MODE=======================================================	
	E_PMLUnitMode.ePMLUnitMode_Maintenance:			
		;	
//	=====================================================================CUSTOM MODE 1==========================================================	
(*	E_PMLUnitMode.ePMLUnitMode_YOURCUSTOMMODE		
		;*)
//	======================================================================INVALID MODE==========================================================	
	E_PMLUnitMode.ePMLUnitMode_Invalid:				
		;
END_CASE
END_METHOD

METHOD Aborting
//bNoStateTasksToComplete := TRUE;		// Change to False if not used

//Implement state Tasks here
(*
IF (insert your completion conditions) THEN

bStateTasksComplete := TRUE;				//Once these actions are completed successfully, set bStateTasksComplete to allow the base code to advance once all children have also reached the proper state

END_IF
*)

SUPER^.Aborting();

(*	Reference State Machine for mode specific actions - Be sure to paste above the SUPER^ Call if used - Delete if not needed

CASE eMode OF
//	====================================================================PRODUCTION MODE=========================================================	
	E_PMLUnitMode.ePMLUnitMode_Production:			
		;
//	====================================================================MANUAL MODE=============================================================	
	E_PMLUnitMode.ePMLUnitMode_Manual:				
		;
//	=====================================================================MAINTENANCE MODE=======================================================	
	E_PMLUnitMode.ePMLUnitMode_Maintenance:			
		;	
//	=====================================================================CUSTOM MODE 1==========================================================	
(*	E_PMLUnitMode.ePMLUnitMode_YOURCUSTOMMODE		
		;*)
//	======================================================================INVALID MODE==========================================================	
	E_PMLUnitMode.ePMLUnitMode_Invalid:				
		;
END_CASE
*)
END_METHOD

METHOD Clearing
//bNoStateTasksToComplete := TRUE;		// Change to False if not used

//Implement state Tasks here
(*
IF (insert your completion conditions) THEN

bStateTasksComplete := TRUE;				//Once these actions are completed successfully, set bStateTasksComplete to allow the base code to advance once all children have also reached the proper state

END_IF
*)

SUPER^.Clearing();
(*	Reference State Machine for mode specific actions - Be sure to paste above the SUPER^ Call if used - Delete if not needed

CASE eMode OF
//	====================================================================PRODUCTION MODE=========================================================	
	E_PMLUnitMode.ePMLUnitMode_Production:			
		;
//	====================================================================MANUAL MODE=============================================================	
	E_PMLUnitMode.ePMLUnitMode_Manual:				
		;
//	=====================================================================MAINTENANCE MODE=======================================================	
	E_PMLUnitMode.ePMLUnitMode_Maintenance:			
		;	
//	=====================================================================CUSTOM MODE 1==========================================================	
(*	E_PMLUnitMode.ePMLUnitMode_YOURCUSTOMMODE		
		;*)
//	======================================================================INVALID MODE==========================================================	
	E_PMLUnitMode.ePMLUnitMode_Invalid:				
		;
END_CASE
*)
END_METHOD

METHOD Complete
CASE eMode OF
//	====================================================================PRODUCTION MODE=========================================================	
	E_PMLUnitMode.ePMLUnitMode_Production:			
		;
//	====================================================================MANUAL MODE=============================================================	
	E_PMLUnitMode.ePMLUnitMode_Manual:				
		;
//	=====================================================================MAINTENANCE MODE=======================================================	
	E_PMLUnitMode.ePMLUnitMode_Maintenance:			
		;	
//	=====================================================================CUSTOM MODE 1==========================================================	
(*	E_PMLUnitMode.ePMLUnitMode_YOURCUSTOMMODE		
		;*)
//	======================================================================INVALID MODE==========================================================	
	E_PMLUnitMode.ePMLUnitMode_Invalid:				
		;
END_CASE
END_METHOD

METHOD Completing
//bNoStateTasksToComplete := TRUE;		// Change to False if not used

//Implement state Tasks here
(*
IF (insert your completion conditions) THEN

bStateTasksComplete := TRUE;				//Once these actions are completed successfully, set bStateTasksComplete to allow the base code to advance once all children have also reached the proper state

END_IF
*)

SUPER^.Completing();

(*	Reference State Machine for mode specific actions - Be sure to paste above the SUPER^ Call if used - Delete if not needed

CASE eMode OF
//	====================================================================PRODUCTION MODE=========================================================	
	E_PMLUnitMode.ePMLUnitMode_Production:			
		;
//	====================================================================MANUAL MODE=============================================================	
	E_PMLUnitMode.ePMLUnitMode_Manual:				
		;
//	=====================================================================MAINTENANCE MODE=======================================================	
	E_PMLUnitMode.ePMLUnitMode_Maintenance:			
		;	
//	=====================================================================CUSTOM MODE 1==========================================================	
(*	E_PMLUnitMode.ePMLUnitMode_YOURCUSTOMMODE		
		;*)
//	======================================================================INVALID MODE==========================================================	
	E_PMLUnitMode.ePMLUnitMode_Invalid:				
		;
END_CASE
*)
END_METHOD

// 
// Cyclic Code
METHOD CyclicLogic
VAR
	i								: UDINT;		//Generic iteration value
END_VAR
// Main loop of the parent module
SUPER^.CyclicLogic();
END_METHOD

METHOD Execute
CASE eMode OF
//	====================================================================PRODUCTION MODE=========================================================	
	E_PMLUnitMode.ePMLUnitMode_Production:			
		;
//	====================================================================MANUAL MODE=============================================================	
	E_PMLUnitMode.ePMLUnitMode_Manual:				
		;
//	=====================================================================MAINTENANCE MODE=======================================================	
	E_PMLUnitMode.ePMLUnitMode_Maintenance:			
		;	
//	=====================================================================CUSTOM MODE 1==========================================================	
(*	E_PMLUnitMode.ePMLUnitMode_YOURCUSTOMMODE		
		;*)
//	======================================================================INVALID MODE==========================================================	
	E_PMLUnitMode.ePMLUnitMode_Invalid:				
		;
END_CASE
END_METHOD

METHOD Held
CASE eMode OF
//	====================================================================PRODUCTION MODE=========================================================	
	E_PMLUnitMode.ePMLUnitMode_Production:			
		;
//	====================================================================MANUAL MODE=============================================================	
	E_PMLUnitMode.ePMLUnitMode_Manual:				
		;
//	=====================================================================MAINTENANCE MODE=======================================================	
	E_PMLUnitMode.ePMLUnitMode_Maintenance:			
		;	
//	=====================================================================CUSTOM MODE 1==========================================================	
(*	E_PMLUnitMode.ePMLUnitMode_YOURCUSTOMMODE		
		;*)
//	======================================================================INVALID MODE==========================================================	
	E_PMLUnitMode.ePMLUnitMode_Invalid:				
		;
END_CASE
END_METHOD

METHOD Holding
//bNoStateTasksToComplete := TRUE;		// Change to False if not used

//Implement state Tasks here
(*
IF (insert your completion conditions) THEN

bStateTasksComplete := TRUE;				//Once these actions are completed successfully, set bStateTasksComplete to allow the base code to advance once all children have also reached the proper state

END_IF
*)

SUPER^.Holding();

(*	Reference State Machine for mode specific actions - Be sure to paste above the SUPER^ Call if used - Delete if not needed

CASE eMode OF
//	====================================================================PRODUCTION MODE=========================================================	
	E_PMLUnitMode.ePMLUnitMode_Production:			
		;
//	====================================================================MANUAL MODE=============================================================	
	E_PMLUnitMode.ePMLUnitMode_Manual:				
		;
//	=====================================================================MAINTENANCE MODE=======================================================	
	E_PMLUnitMode.ePMLUnitMode_Maintenance:			
		;	
//	=====================================================================CUSTOM MODE 1==========================================================	
(*	E_PMLUnitMode.ePMLUnitMode_YOURCUSTOMMODE		
		;*)
//	======================================================================INVALID MODE==========================================================	
	E_PMLUnitMode.ePMLUnitMode_Invalid:				
		;
END_CASE
*)
END_METHOD

METHOD Idle
CASE eMode OF
//	====================================================================PRODUCTION MODE=========================================================	
	E_PMLUnitMode.ePMLUnitMode_Production:			
		;
//	====================================================================MANUAL MODE=============================================================	
	E_PMLUnitMode.ePMLUnitMode_Manual:				
		;
//	=====================================================================MAINTENANCE MODE=======================================================	
	E_PMLUnitMode.ePMLUnitMode_Maintenance:			
		;	
//	=====================================================================CUSTOM MODE 1==========================================================	
(*	E_PMLUnitMode.ePMLUnitMode_YOURCUSTOMMODE		
		;*)
//	======================================================================INVALID MODE==========================================================	
	E_PMLUnitMode.ePMLUnitMode_Invalid:				
		;
END_CASE
END_METHOD

METHOD Initialize
VAR
	i								: UDINT;		//Generic iteration value
END_VAR

// Define the interfaces to the different subunits (Must take place before SUPER^.initialize call)
FOR i := 1 TO MAX_NO_OF_SUBMODULES DO
	a_ITF_PackMLBase[i] := a_ITF_PackMLBase_init[i];
END_FOR

FOR i := 1 TO MAX_NO_OF_COMPONENTS DO
	a_ITF_Components[i] := a_ITF_Components_init[i];
END_FOR

// Init of the parent class object (Must be called AFTER most local init code, since the sub module interface array assignments should be made here, and then operated on within the module base init
SUPER^.Initialize();
END_METHOD

METHOD Resetting
//bNoStateTasksToComplete := TRUE;		// Change to False if not used

//Implement state Tasks here
(*
IF (insert your completion conditions) THEN

bStateTasksComplete := TRUE;				//Once these actions are completed successfully, set bStateTasksComplete to allow the base code to advance once all children have also reached the proper state

END_IF
*)

SUPER^.Resetting();

(*	Reference State Machine for mode specific actions - Be sure to paste above the SUPER^ Call if used - Delete if not needed

CASE eMode OF
//	====================================================================PRODUCTION MODE=========================================================	
	E_PMLUnitMode.ePMLUnitMode_Production:			
		;
//	====================================================================MANUAL MODE=============================================================	
	E_PMLUnitMode.ePMLUnitMode_Manual:				
		;
//	=====================================================================MAINTENANCE MODE=======================================================	
	E_PMLUnitMode.ePMLUnitMode_Maintenance:			
		;	
//	=====================================================================CUSTOM MODE 1==========================================================	
(*	E_PMLUnitMode.ePMLUnitMode_YOURCUSTOMMODE		
		;*)
//	======================================================================INVALID MODE==========================================================	
	E_PMLUnitMode.ePMLUnitMode_Invalid:				
		;
END_CASE
*)
END_METHOD

METHOD Starting
//bNoStateTasksToComplete := TRUE;		// Change to False if not used

//Implement state Tasks here
(*
IF (insert your completion conditions) THEN

bStateTasksComplete := TRUE;				//Once these actions are completed successfully, set bStateTasksComplete to allow the base code to advance once all children have also reached the proper state

END_IF
*)

SUPER^.Starting();

(*	Reference State Machine for mode specific actions - Be sure to paste above the SUPER^ Call if used - Delete if not needed

